VAR
	pRack 		: POINTER TO FB_Rack;
	pReactor 	: POINTER TO FB_Reactor;
	pNeedle		: POINTER TO FB_Needle; 
	pSlot 		: POINTER TO FB_PieceSlot;
	pTarget 	: POINTER TO FB_TargetBase;
	pPieceEx	: POINTER TO FB_PieceBase;
END_VAR
CASE refActionData.eAction OF
	E_Action.ACTION_ExchangePiece:
		pTarget := fbObjectDirectory.M_GetObjPointer(refActionData.nTarget);
		//Piece, welches gehandelt wird
		pPieceEx := pCorrelObject;
		//Welches Piece soll gehandelt werden?
		IF refActionData.aParams[2] = 0 THEN //Drop
			IF pPiece = 0 THEN
				M_CheckAction := E_ErrorIdCmd.ERRORID_NoPieceOnTool;
				RETURN;	
			END_IF
			//Luer kann folgende Pieces handeln
			//Tip, Needle, Septum in Verbindung mit Needle
			IF pPiece^.P_eObjectType = E_ObjectType.OBJECTTYPE_Tip THEN
				//Target muss TipRack sein
				IF pTarget^.P_eObjectType <> E_ObjectType.OBJECTTYPE_TipRack THEN
					M_CheckAction := E_ErrorIdCmd.ERRORID_UnsuitableTarget;
					RETURN;
				END_IF
			ELSIF pPiece^.P_eObjectType = E_ObjectType.OBJECTTYPE_Needle THEN
				pNeedle := pPiece;
				IF pNeedle^.P_pSeptum > 0 THEN
					//Target muss SeptumWaste sein
					IF pTarget^.P_eObjectType <> E_ObjectType.OBJECTTYPE_SeptumWaste THEN
						M_CheckAction := E_ErrorIdCmd.ERRORID_UnsuitableTarget;
						RETURN;
					END_IF
				ELSE
					//Target muss NeedleRack sein
					IF pTarget^.P_eObjectType <> E_ObjectType.OBJECTTYPE_NeedleRack THEN
						M_CheckAction := E_ErrorIdCmd.ERRORID_UnsuitableTarget;
						RETURN;
					END_IF
				END_IF
			ELSE
				M_CheckAction := E_ErrorIdCmd.ERRORID_InvalidPieceType;
				RETURN;
			END_IF
		ELSE //Take
			//Schon ein Piece am Tool?
			IF pPiece > 0 THEN
				IF pPiece^.P_eObjectType = E_ObjectType.OBJECTTYPE_Needle THEN
					pNeedle := pPiece;
					IF pNeedle^.P_pSeptum > 0 THEN
						M_CheckAction := E_ErrorIdCmd.ERRORID_PieceAlreadyOnTool;
						RETURN;
					ELSE
						//Target muss Reactor sein!
						IF pTarget^.P_eObjectType = E_ObjectType.OBJECTTYPE_Reactor THEN
							//Im Reaktor muss ein Vial und auf diesem sich ein Septum befinden
							pReactor := pTarget;
							IF pReactor^.P_pVial > 0 THEN
								IF pReactor^.P_pVial^.P_pSeptum = 0 THEN
									M_CheckAction := E_ErrorIdCmd.ERRORID_NoPieceInSlot;
									RETURN;
								END_IF
							ELSE
								M_CheckAction := E_ErrorIdCmd.ERRORID_NoPieceInSlot;
								RETURN;
							END_IF
						ELSE
							M_CheckAction := E_ErrorIdCmd.ERRORID_UnsuitableTarget;
							RETURN;
						END_IF
					END_IF
				ELSE
					M_CheckAction := E_ErrorIdCmd.ERRORID_PieceAlreadyOnTool;
					RETURN;
				END_IF
			ELSE 
				IF pPieceEx^.P_eObjectType = E_ObjectType.OBJECTTYPE_Septum THEN
					M_CheckAction := E_ErrorIdCmd.ERRORID_NoNeedleOnTool;
					RETURN;
				END_IF
			END_IF
		END_IF	
	E_Action.ACTION_DockTool:
		pTarget := fbObjectDirectory.M_GetObjPointer(refActionData.nTarget);
		//Piece am Tool?
		IF THIS^.pPiece > 0 THEN
			M_CheckAction := E_ErrorIdCmd.ERRORID_PieceAlreadyOnTool;
			RETURN;
		END_IF
		//Luer kann an PortRack andocken
		IF pTarget^.P_eObjectType = E_ObjectType.OBJECTTYPE_PortRack THEN
			pRack := pTarget;
			pSlot := pRack^.M_GetSlot(DINT_TO_UINT(refActionData.aParams[2]));
			IF pSlot > 0 THEN
				IF pSlot^.P_pPiece = 0 THEN
					M_CheckAction := E_ErrorIdCmd.ERRORID_NoPieceInSlot;
					RETURN;	
				END_IF
			ELSE
				M_CheckAction := E_ErrorIdCmd.ERRORID_InvalidTargetSlot;
				RETURN;
			END_IF
			//Im Slot muss ein Port sein
		ELSE
			M_CheckAction := E_ErrorIdCmd.ERRORID_UnsuitableTarget;
			RETURN;		
		END_IF
	E_Action.ACTION_MeasureTool:
		IF fbObjectDirectory.M_GetObjType(refActionData.nTarget) <> E_ObjectType.OBJECTTYPE_TipCalibrator THEN
			M_CheckAction := E_ErrorIdCmd.ERRORID_UnsuitableTarget;
			RETURN;
		END_IF
	E_Action.ACTION_InsertTool:
		IF pPiece = 0 THEN
			M_CheckAction := E_ErrorIdCmd.ERRORID_NoPieceOnTool;
		END_IF
	E_Action.ACTION_WashTool:
		//Washmode checken
		IF refActionData.aParams[2] = E_WashMode.MODE_WashInside THEN
			M_CheckAction := M_CheckBottles();
		ELSIF refActionData.aParams[2] = E_WashMode.MODE_WashOutside THEN
			;
		ELSIF refActionData.aParams[2] = E_WashMode.MODE_WashInOutside THEN
			M_CheckAction := M_CheckBottles();
		ELSE
			M_CheckAction := E_ErrorIdCmd.ERRORID_InvalidWashMode;	
		END_IF	
	E_Action.ACTION_Dispense, //BasicAction für ActionOnArray
	E_Action.ACTION_DryToolInside,
	E_Action.ACTION_TeachTarget:
		RETURN;
ELSE
	M_CheckAction := SUPER^.M_CheckAction(refActionData, pCorrelObject);
END_CASE
END_METHOD

METHOD M_CheckBottles : ERRORID
VAR_INPUT
END_VAR
IF pDiluter > 0 THEN
	M_CheckBottles := pDiluter^.M_CheckBottles(0);
END_IF
END_METHOD

METHOD M_CheckProps : ERRORID
VAR_INPUT
END_VAR
M_CheckProps := SUPER^.M_CheckProps();
IF M_CheckProps > 0 THEN
	RETURN;
END_IF
//Konfigurierte Properties checken
//zugeordneter Diluter
IF fbObjectDirectory.M_GetObjType(nDiluterObjId) <> E_ObjectType.OBJECTTYPE_Diluter THEN
	M_CheckProps := E_ErrorIdObjMgmt.ERRORID_InvalidDiluterObjId; //Error
	RETURN;
ELSE
	pDiluter := fbObjectDirectory.M_GetObjPointer(nDiluterObjId);
END_IF
END_METHOD

METHOD M_ClearAllProps
VAR_INPUT
	bIgnoreParent : BOOL; //Es wird das gesamte OD gelöscht. -> Zeiger auf Parent nicht mehr gültig!
END_VAR
pPneuChannelSyntGas := 0;
SUPER^.M_ClearAllProps(bIgnoreParent);
END_METHOD

METHOD M_ExeAction : ERRORID
VAR_INPUT
	refActionData : REFERENCE TO ST_ActionData;	
END_VAR
IF NOT (eCurrentState = E_MachineState.MACHINESTATE_Idle OR
	eCurrentState = E_MachineState.MACHINESTATE_Active OR
	eCurrentState = E_MachineState.MACHINESTATE_Ready) THEN
	M_ExeAction := E_ErrorIdCmd.ERRORID_InvalidState;
	RETURN;
END_IF

CASE refActionData.eAction OF
	
	E_Action.ACTION_Aspirate:
		IF NOT bAspirate THEN
			M_ExeAction := pDiluter^.M_CheckBottles(0); //Checken, ob Bottles OK
			IF M_ExeAction > 0 THEN
				RETURN;
			END_IF			
			nQuantity := refActionData.aParams[1];
			nFlow := refActionData.aParams[2];
			fbList.A_AddHeadValue( hList := hList, putValue := E_Action.ACTION_Aspirate);
			bAspirate := TRUE;
		END_IF
		
	E_Action.ACTION_Dispense:
		IF NOT bDispense THEN
			M_ExeAction := pDiluter^.M_CheckBottles(0); //Checken, ob Bottles OK
			IF M_ExeAction > 0 THEN
				RETURN;
			END_IF			
			nQuantity := refActionData.aParams[1];
			nFlow := refActionData.aParams[2];
			fbList.A_AddHeadValue(hList := hList, putValue := E_Action.ACTION_Dispense);
			bDispense := TRUE;
		END_IF
		
	E_Action.ACTION_Mix:
		IF NOT bMix THEN
			M_ExeAction := pDiluter^.M_CheckBottles(0); //Checken, ob Bottles OK
			IF M_ExeAction > 0 THEN
				RETURN;
			END_IF			
			nQuantity := refActionData.aParams[1];
			nFlowAsp := refActionData.aParams[2];
			nFlowDisp := refActionData.aParams[3];
			nMixRepeats := DINT_TO_UINT(refActionData.aParams[4]);
			nCurrMixRepeats := 0;
			tMixDelay1 := DINT_TO_TIME(refActionData.aParams[5]);
			tMixDelay2 := DINT_TO_TIME(refActionData.aParams[6]);
			fbList.A_AddHeadValue(hList := hList, putValue := E_Action.ACTION_Mix);
			bMix := TRUE;
		END_IF		
		
	E_Action.ACTION_Eject:
		//TipEjector vorhanden??
		IF pZAxisRef^.eFixedToolType <> E_MzToolType.TOOL_TYPE_TipEjector THEN
			M_ExeAction := 21212;
			RETURN;	
		END_IF
		
		IF NOT bEject THEN
			fbList.A_AddHeadValue(hList := hList, putValue := E_Action.ACTION_Eject);
			bEject := TRUE;
		END_IF
			
	E_Action.ACTION_SetPressure:
		fbSetPress(bExecute:= FALSE, pPneuChannelRef:= pPneuChannelSyntGas); //eventueller Fehler wird auch zurückgesetzt
		fbSetPress.bAwait := DINT_TO_BOOL(refActionData.aParams[1]);
		fbSetPress.nValue := DINT_TO_INT(refActionData.aParams[2]);
		fbSetPress.nTolerancePlus := DINT_TO_INT(refActionData.aParams[3]);
		fbSetPress.nToleranceMinus := DINT_TO_INT(refActionData.aParams[4]);
		fbSetPress.tTimeout := DINT_TO_TIME(refActionData.aParams[5]);
		
		fbSetPress(bExecute:= TRUE,	pPneuChannelRef:= pPneuChannelSyntGas, nErrorId=> M_ExeAction);
		IF fbSetPress.bError THEN
			RETURN;
		END_IF
		
		IF NOT bSetPress AND fbSetPress.bBusy THEN
			bSetPress := TRUE;
			fbList.A_AddHeadValue(hList := hList, putValue := E_Action.ACTION_SetPressure);
		ELSE
			RETURN;	
		END_IF
		
	E_Action.ACTION_SwitchPressure:
		eSwitchPressCtrl := DINT_TO_USINT(refActionData.aParams[1]);
		tPressTime := DINT_TO_TIME(refActionData.aParams[2]);
		//Wenn Aktion aktiv kann es sein das die Zeit noch läuft oder der Druck an ist
		IF bSwitchPress THEN	//Aktion ist aktiv
			IF eSwitchPressCtrl = E_PressCtrl.PRESSCTRL_PressOn THEN
				//Statemachine zurücksetzen
				nStateA_SwitchPress := 0;		
			ELSE
				aValves[nValveNrSynthGas].M_Off();
				nStateA_SwitchPress := 80;
			END_IF
		ELSE	//Aktion ist nicht aktiv
			IF eSwitchPressCtrl = E_PressCtrl.PRESSCTRL_PressOn THEN
				bSwitchPress := TRUE;
				fbList.A_AddHeadValue(hList := hList, putValue := E_Action.ACTION_SwitchPressure);
			ELSE
				aValves[nValveNrSynthGas].M_Off();
			END_IF
		END_IF
	ELSE
		M_ExeAction := SUPER^.M_ExeAction(refActionData);
		RETURN;
END_CASE

bBusy := TRUE;
eCurrentState := E_MachineState.MACHINESTATE_Active;
END_METHOD

METHOD M_GetAllProps : ERRORID
VAR_INPUT
	refCmdData : REFERENCE TO  ST_CmdData;
END_VAR
//BaseProperties lesen
SUPER^.M_GetAllProps(refCmdData);
//BaseProperties lesen
nCurrentPropIndex := nCurrentPropIndex + 1;
refCmdData.n32Data[nCurrentPropIndex] := nDiluterObjId;
nCurrentPropIndex := nCurrentPropIndex + 1;
refCmdData.n32Data[nCurrentPropIndex] := nDiluterObjId2;
nCurrentPropIndex := nCurrentPropIndex + 1;
refCmdData.n32Data[nCurrentPropIndex] := nDrypadArea;
nCurrentPropIndex := nCurrentPropIndex + 1;
refCmdData.n32Data[nCurrentPropIndex] := TIME_TO_DINT(tDryTime);
//TipEjector exist
nCurrentPropIndex := nCurrentPropIndex + 1;
IF pZAxisRef^.eFixedToolType = E_MzToolType.TOOL_TYPE_TipEjector THEN
	refCmdData.n32Data[nCurrentPropIndex] := 1;
ELSE
	refCmdData.n32Data[nCurrentPropIndex] := 0;
END_IF

nCurrentPropIndex := nCurrentPropIndex + 1;
IF pPneuChannelSyntGas > 0 THEN
	refCmdData.n32Data[nCurrentPropIndex] := pPneuChannelSyntGas^.nChannel;	
ELSE
	refCmdData.n32Data[nCurrentPropIndex] := 0;
END_IF

nCurrentPropIndex := nCurrentPropIndex + 1;
refCmdData.n32Data[nCurrentPropIndex] := nValveNrSynthGas;
nCurrentPropIndex := nCurrentPropIndex + 1;
refCmdData.n32Data[nCurrentPropIndex] := nValveNrDiluter;
nCurrentPropIndex := nCurrentPropIndex + 1;
refCmdData.n32Data[nCurrentPropIndex] := nValveNrLuer;
nCurrentPropIndex := nCurrentPropIndex + 1;
refCmdData.n32Data[nCurrentPropIndex] := REAL_TO_DINT(rDockOffset);
nCurrentPropIndex := nCurrentPropIndex + 1;
refCmdData.n32Data[nCurrentPropIndex] := nDispFlowFix;
END_METHOD

METHOD M_SetAllProps : ERRORID
VAR_INPUT
	refCmdData : REFERENCE TO  ST_CmdData;
END_VAR

VAR
	nPneuChannel : USINT;
END_VAR
M_SetAllProps := SUPER^.M_SetAllProps(refCmdData);

IF M_SetAllProps > 0 THEN
	RETURN;
END_IF

//Diluter 1 (SingleDiluter)
nCurrentPropIndex := nCurrentPropIndex + 1;
nSpecPropIndex := nCurrentPropIndex;
nDiluterObjId :=  DINT_TO_UINT(refCmdData.n32Data[nCurrentPropIndex]);

IF fbObjectDirectory.M_GetObjType(nDiluterObjId) = E_ObjectType.OBJECTTYPE_Diluter THEN
	pDiluter := fbObjectDirectory.M_GetObjPointer(nDiluterObjId);
ELSE
	M_SetAllProps := E_ErrorIdObjMgmt.ERRORID_InvalidDiluterObjId;
	RETURN;
END_IF

//Diluter 2 (TwinDiluter)
nCurrentPropIndex := nCurrentPropIndex + 1;
nDiluterObjId2 :=  DINT_TO_UINT(refCmdData.n32Data[nCurrentPropIndex]);

nCurrentPropIndex := nCurrentPropIndex + 1;
nDrypadArea := DINT_TO_USINT(refCmdData.n32Data[nCurrentPropIndex]);
nCurrentPropIndex := nCurrentPropIndex + 1;
tDryTime := DINT_TO_TIME(refCmdData.n32Data[nCurrentPropIndex]);

//TipEjector
nCurrentPropIndex := nCurrentPropIndex + 1;
IF refCmdData.n32Data[nCurrentPropIndex].0 THEN
	pZAxisRef^.eFixedToolType := E_MzToolType.TOOL_TYPE_TipEjector;
ELSE
	pZAxisRef^.eFixedToolType := E_MzToolType.TOOL_TYPE_None;
END_IF

nCurrentPropIndex := nCurrentPropIndex + 1;
nPneuChannel := DINT_TO_USINT(refCmdData.n32Data[nCurrentPropIndex]);
IF NOT (nPneuChannel > 0 AND nPneuChannel <= cNoOfPneuChannels) THEN
	M_SetAllProps := E_ErrorIdObjMgmt.ERRORID_InvalidPneuChannel;
	RETURN;
END_IF
pPneuChannelSyntGas := ADR(aFbPneuChannel[nPneuChannel]);

nCurrentPropIndex := nCurrentPropIndex + 1;
nValveNrSynthGas := DINT_TO_USINT(refCmdData.n32Data[nCurrentPropIndex]);
IF NOT(nValveNrSynthGas >= 0 AND nValveNrSynthGas <= cNoOfValves) THEN
	M_SetAllProps := E_ErrorIdObjMgmt.ERRORID_InvalidValveNumber;
	RETURN;
END_IF

nCurrentPropIndex := nCurrentPropIndex + 1;
nValveNrDiluter := DINT_TO_USINT(refCmdData.n32Data[nCurrentPropIndex]);
IF NOT(nValveNrDiluter >= 0 AND nValveNrDiluter <= cNoOfValves) THEN
	M_SetAllProps := E_ErrorIdObjMgmt.ERRORID_InvalidValveNumber;
END_IF

nCurrentPropIndex := nCurrentPropIndex + 1;
nValveNrLuer := DINT_TO_USINT(refCmdData.n32Data[nCurrentPropIndex]);
IF NOT(nValveNrLuer >= 0 AND nValveNrLuer <= cNoOfValves) THEN
	M_SetAllProps := E_ErrorIdObjMgmt.ERRORID_InvalidValveNumber;
END_IF

nCurrentPropIndex := nCurrentPropIndex + 1;
rDockOffset := DINT_TO_REAL(refCmdData.n32Data[nCurrentPropIndex]);

//DispFlowFix
nCurrentPropIndex := nCurrentPropIndex + 1;
nDispFlowFix := refCmdData.n32Data[nCurrentPropIndex];

nNoOfProps := nCurrentPropIndex + 1;
END_METHOD

METHOD M_SetPrintParams : ST_MethResult
VAR_INPUT
	eType 		: E_PrintParamType;
	nNumerator	: USINT;
	nValue		: DINT;
END_VAR
IF eType = E_PrintParamType.Flow THEN
	IF nNumerator <> 1 THEN
		M_SetPrintParams.bError := TRUE;
		M_SetPrintParams.nErrorId := E_ErrorIdCmd.ERRORID_InvalidPrintParamNumerator;
		RETURN;
	END_IF
	fbObjectDirectory.M_SetObjChange(nObjectID); //Info an GUI
	nDispFlowFix := nValue;
ELSE
	M_SetPrintParams.bError := TRUE;
	M_SetPrintParams.nErrorId := E_ErrorIdCmd.ERRORID_InvalidPrintParamType;
END_IF
END_METHOD

METHOD M_SetSingleProp : ERRORID
VAR_INPUT
	refCmdData : REFERENCE TO  ST_CmdData;
END_VAR

VAR
	nPneuChannel : USINT;
END_VAR
IF nSpecPropIndex + 5 = refCmdData.aHeader[1] THEN	//PneuChannelSynthGas
	nPneuChannel := DINT_TO_USINT(refCmdData.n32Data[0]);
	IF NOT (nPneuChannel > 0 AND nPneuChannel <= cNoOfPneuChannels) THEN
		M_SetSingleProp := E_ErrorIdObjMgmt.ERRORID_InvalidPneuChannel;
		RETURN;	
	END_IF
	pPneuChannelSyntGas := ADR(aFbPneuChannel[nPneuChannel]);
ELSIF nSpecPropIndex + 6 = refCmdData.aHeader[1] THEN	//ValveSynthGas
	IF refCmdData.n32Data[0] >= 0 AND refCmdData.n32Data[0] <= cNoOfValves THEN
		nValveNrSynthGas := DINT_TO_USINT(refCmdData.n32Data[0]);
	ELSE
		M_SetSingleProp := E_ErrorIdObjMgmt.ERRORID_InvalidValveNumber;
	END_IF
ELSIF nSpecPropIndex + 7 = refCmdData.aHeader[1] THEN	//ValveNrDiluter
	IF refCmdData.n32Data[0] >= 0 AND refCmdData.n32Data[0] <= cNoOfValves THEN
		nValveNrDiluter := DINT_TO_USINT(refCmdData.n32Data[0]);
	ELSE
		M_SetSingleProp := E_ErrorIdObjMgmt.ERRORID_InvalidValveNumber;
	END_IF	
ELSIF nSpecPropIndex + 8 = refCmdData.aHeader[1] THEN	//ValveNrLuer
	IF refCmdData.n32Data[0] >= 0 AND refCmdData.n32Data[0] <= cNoOfValves THEN
		nValveNrLuer := DINT_TO_USINT(refCmdData.n32Data[0]);
	ELSE
		M_SetSingleProp := E_ErrorIdObjMgmt.ERRORID_InvalidValveNumber;
	END_IF	
ELSIF nSpecPropIndex + 9 = refCmdData.aHeader[1] THEN	//DockOffset
	rDockOffset := DINT_TO_REAL(refCmdData.n32Data[0]);
ELSIF nSpecPropIndex + 10 = refCmdData.aHeader[1] THEN	//DispFlowFix
	nDispFlowFix := refCmdData.n32Data[0];
ELSE
	M_SetSingleProp := SUPER^.M_SetSingleProp(refCmdData);
END_IF
END_METHOD

METHOD M_StartUniDispense : ERRORID
VAR_INPUT
	nParam1 : DINT; //Quantity
	nParam2 : DINT; //unused
END_VAR

VAR_OUTPUT
	bIsContinous : BOOL;
END_VAR

VAR
	stActionData : ST_ActionData;
END_VAR
IF nParam1 = 0 THEN
	bIsContinous := TRUE;
	bEndless := TRUE;
ELSE
	bEndless := FALSE;
END_IF

stActionData.aParams[1] := nParam1; //Quantitiy
stActionData.aParams[2] := nDispFlowFix;
stActionData.eAction := E_Action.ACTION_Dispense;
M_StartUniDispense := M_ExeAction(stActionData);
END_METHOD

METHOD M_StopUniDispense : ERRORID
VAR_INPUT
END_VAR
M_CancelAction(E_Action.ACTION_Dispense);
END_METHOD

METHOD M_SwitchValveDiluter
VAR_INPUT
	bOn : BOOL;
END_VAR
IF nValveNrDiluter > 0 THEN
	IF bOn THEN
		aValves[nValveNrDiluter].M_On(1);
	ELSE
		aValves[nValveNrDiluter].M_Off();
	END_IF
END_IF
END_METHOD

METHOD M_SwitchValveLuer
VAR_INPUT
	bOn : BOOL;
END_VAR
IF nValveNrLuer > 0 THEN
	IF bOn THEN
		aValves[nValveNrLuer].M_On(1);
	ELSE
		aValves[nValveNrLuer].M_Off();
	END_IF
END_IF
END_METHOD

METHOD M_SwitchValveSynthGas
VAR_INPUT
	bOn : BOOL;
END_VAR
IF nValveNrSynthGas > 0 THEN
	IF bOn THEN
		aValves[nValveNrSynthGas].M_On(1);
	ELSE
		aValves[nValveNrSynthGas].M_Off();
	END_IF
END_IF
END_METHOD

PROPERTY P_nDrypadArea : USINT
GET
P_nDrypadArea := nDrypadArea;
END_GET
END_PROPERTY

PROPERTY P_pDiluter : POINTER TO FB_DILUTER
GET
P_pDiluter := pDiluter;
END_GET
END_PROPERTY

PROPERTY P_rDockOffset : REAL
GET
P_rDockOffset := rDockOffset;
END_GET
END_PROPERTY

PROPERTY P_stAbsPosPhys : ST_3DPoint
GET
VAR
	stTemp	: ST_3DPoint;
	stDim	: ST_3DDimension;
END_VAR
//Die absolute Postion eines Tool in "Z" hat nicht den gleichen Bezug wie X und Y
//X und Y beziehen sich auf den Koordinatenursprung, wenn die Achsen theoretischn aus Antrieb (0;0) stehen
//Z bezieht sich auf die Sliderunterkante des Z-Antriebes verechnet mit AbsPos vom Head(Ergebnis ist in den meisten Fällen negativ)

//Offset und RelPos addieren
stTemp := F_Add3DPoints(stRelPos,stOffset);

//Offsets der Pieces verrechnen
IF pPiece > 0 THEN
	stDim := pPiece^.P_stDimension;
	IF NOT pPiece^.P_bIgnoreOffset THEN
		stTemp := F_Add3DPoints(stTemp,pPiece^.P_stOffset);	
	END_IF
	stTemp.Z := stTemp.Z + pPiece^.P_rZOverlapTool - stDim.Height;
END_IF

//AbsPos vom ParentSlot holen
IF pParentSlot > 0 THEN
	stTemp := F_Add3DPoints(stTemp,pParentSlot^.P_stAbsPos);	
END_IF
P_stAbsPosPhys := stTemp;
END_GET
END_PROPERTY

PROPERTY P_stCurrentXYArea : FB_RectAngle
GET
VAR
	stPoint : ST_3DPoint;
	stDim	: ST_3DDimension;
END_VAR
stPoint := P_stCurrentPosPhys;
IF pPiece > 0 THEN
	stDim := pPiece^.P_stDimension;
	P_stCurrentXYArea.X1 := stPoint.X - stDim.Width / 2.0;
	P_stCurrentXYArea.X2 := stPoint.X + stDim.Width / 2.0;
	P_stCurrentXYArea.Y1 := stPoint.Y - stDim.Width / 2.0;
	P_stCurrentXYArea.Y2 := stPoint.Y + stDim.Width / 2.0;
ELSE
	P_stCurrentXYArea.X1 := stPoint.X - 2000.0;
	P_stCurrentXYArea.X2 := stPoint.X + 2000.0;
	P_stCurrentXYArea.Y1 := stPoint.Y - 2000.0;
	P_stCurrentXYArea.Y2 := stPoint.Y + 2000.0;	
END_IF
END_GET
END_PROPERTY

PROPERTY P_tDryTime : TIME
GET
P_tDryTime := tDryTime;
END_GET
END_PROPERTY

END_FUNCTION_BLOCK

// ---- Objects/Tools/FB_VacuumHandler.TcPOU
FUNCTION_BLOCK FB_VacuumHandler EXTENDS FB_MzTool
VAR_INPUT
END_VAR
VAR_OUTPUT
END_VAR
VAR
	

	//SpecProperties
	pPneuChannelVac		: POINTER TO FB_PneuChannelRef;
	nValveNrVacuum		: USINT;
	nHoldVacuumVial		: INT;
	nHoldVacuumSeptum	: INT;
	rDockOffset			: REAL;

	//****************************************Aktionvariablen****************************************************
	
	stActionDataSpec	: ST_ActionData;
	
	//Action: "InitSpec"
	bInitSpec			: BOOL;
	bInitSpecFlag		: BOOL := TRUE;
	nStateA_InitSpec	: USINT;
	
	//Action: "SetVacuum"
	bSetVacuum			: BOOL;
	fbSetVacuum			: FB_SetPressure;
	
	//Action: "SwitchPressure"
	bSwitchPress		: BOOL;			
	nStateA_SwitchPress	: USINT;		//State von A_SwitchPress()
	nSwitchPressChannel	: USINT;
	eSwitchPressCtrl	: E_PressCtrl;
	tPressTime			: TIME;			//nach dieser Zeit Ventil automatisch wieder zu
	timerPress			: TON;			//Timer für Öffnungszeit Druckventil 		
	
END_VAR

IF eCurrentState = E_MachineState.MACHINESTATE_Active THEN
	
	IF bSetVacuum THEN
		fbSetVacuum(pPneuChannelRef:= pPneuChannelVac);
		IF NOT fbSetVacuum.bBusy THEN
			IF fbSetVacuum.bError THEN
				bError := TRUE;
				stError.ErrorId := fbSetVacuum.nErrorId;
				stError.POU := E_POU.POU_FB_VacuumHandler;
				fbErrorList.M_Add(stError);
			END_IF
			bSetVacuum := FALSE;
			fbSetVacuum(pPneuChannelRef:= pPneuChannelVac, bExecute:= FALSE);
			M_RemoveListEntry(nSearchValue:= E_Action.ACTION_SetVacuum);
		END_IF
	END_IF	
	
	IF bSwitchPress THEN	//Kartuschendruck einstellen und Ein-bzw. Aus schalten 
		A_SwitchPress();
		IF nStateA_SwitchPress >= 80 THEN
			IF nStateA_SwitchPress >= 99 THEN
				bError := TRUE;
			END_IF
			bSwitchPress := FALSE;
			nStateA_SwitchPress := 0;
			M_RemoveListEntry(nSearchValue:= E_Action.ACTION_SwitchPressure);
		END_IF
	END_IF	
END_IF

SUPER^();	//FB_MzTool aufrufen

//Prozessdaten aktualisieren
IF pPneuChannelVac > 0 THEN
	stProcessData.n32Data[7] := pPneuChannelVac^.P_nCurrentPressure;
END_IF

IF nValveNrVacuum > 0 THEN
	IF aValves[nValveNrVacuum].bDigiOut1 THEN
		stProcessData.n32Data[8] := E_PressCtrl.PRESSCTRL_VacOn;
	ELSE
		stProcessData.n32Data[8] := E_PressCtrl.PRESSCTRL_Off;
	END_IF
END_IF

aObjProcData[nNotifyId] := stProcessData;

ACTION A_Reset:
//Ist noch eine Aktion aktiv?
IF nStateA_ResetSpec = 0 THEN 
	nStateA_ResetSpec := 80;
END_IF

SUPER^.A_Reset();
END_ACTION

ACTION A_Stop:
IF nStateA_Stop = 0 THEN
	nStateA_Stop := 1;
END_IF

SUPER^.A_Stop();
END_ACTION

ACTION A_SwitchPress:
CASE nStateA_SwitchPress OF
	0:	//Ventil Einschalten
		IF eSwitchPressCtrl = E_PressCtrl.PRESSCTRL_PressOn OR eSwitchPressCtrl = E_PressCtrl.PRESSCTRL_VacOn THEN
			aValves[M_GetValveNr(nSwitchPressChannel)].M_On(1);
		END_IF
	
		//Timer starten
		IF tPressTime = T#0S THEN
			nStateA_SwitchPress := 80;
			RETURN;	
		END_IF
		
		timerPress(IN:= FALSE);
		timerPress(IN:= TRUE, PT:= tPressTime);
		nStateA_SwitchPress := 1;
		
	1:	//Warten bis Zeitabgelaufen
		timerPress();
		IF timerPress.Q THEN
			timerPress(IN:= FALSE);
			aValves[M_GetValveNr(nSwitchPressChannel)].M_Off();
			nStateA_SwitchPress := 80;
		END_IF
		
	70:	//Abbrechen
		timerPress(IN:= FALSE);
		aValves[M_GetValveNr(nSwitchPressChannel)].M_Off();
		nStateA_SwitchPress := 80;
END_CASE
END_ACTION

METHOD FB_init : BOOL
VAR_INPUT
	bInitRetains : BOOL; // if TRUE, the retain variables are initialized (warm start / cold start)
	bInCopyCode : BOOL;  // if TRUE, the instance afterwards gets moved into the copy code (online change)
END_VAR
eObjectType := E_ObjectType.OBJECTTYPE_VacuumHandler;
eObjectGroup := E_ObjectGroup.OBJECTGROUP_MzTool OR E_ObjectGroup.OBJECTGROUP_Device;
END_METHOD

METHOD M_AddChild : ERRORID
VAR_INPUT
	pObject : POINTER TO FB_Object;
	nSlotNr	: UINT;
	nIndex 	: INT;	
END_VAR
//Kann folgende Objekt-Typen aufnehmen
//Vial, Septum
IF pObject > 0 THEN
	IF pObject^.P_eObjectType = E_ObjectType.OBJECTTYPE_Vial OR
		pObject^.P_eObjectType = E_ObjectType.OBJECTTYPE_Septum THEN
		M_AddChild := SUPER^.M_AddChild(pObject,nSlotNr,nIndex);
	ELSE
		M_AddChild := E_ErrorIdObjMgmt.ERRORID_InvalidParentObject;
	END_IF
ELSE
	M_AddChild := E_ErrorIdObjMgmt.ERRORID_InvalidParentObject;
END_IF
END_METHOD

METHOD M_CancelAction
VAR_INPUT
	eAction : E_Action;
END_VAR
CASE eAction OF

	E_Action.ACTION_SetVacuum:
		IF bSetVacuum THEN
			fbSetVacuum(bExecute:= FALSE, pPneuChannelRef:= pPneuChannelVac);
		END_IF

	E_Action.ACTION_SwitchPressure:
		IF bSwitchPress AND nStateA_SwitchPress < 70 THEN
			nStateA_SwitchPress := 70;
		END_IF	
ELSE
	SUPER^.M_CancelAction(eAction);
END_CASE
END_METHOD

METHOD M_CheckAction : ERRORID
VAR_INPUT
	refActionData 	: REFERENCE TO ST_ActionData;
	pCorrelObject	: POINTER TO FB_Object;
END_VAR

VAR
	pRack : POINTER TO FB_Rack;
	pReactor : POINTER TO FB_Reactor;
	pSlot : POINTER TO FB_PieceSlot;
	pTarget : POINTER TO FB_TargetBase;
END_VAR
CASE refActionData.eAction OF
	E_Action.ACTION_ExchangePiece:
		pTarget := fbObjectDirectory.M_GetObjPointer(refActionData.nTarget);
		//Welches Piece soll gehandelt werden?
		IF refActionData.aParams[2] = 0 THEN //Drop
			IF pPiece = 0 THEN
				M_CheckAction := E_ErrorIdCmd.ERRORID_NoPieceOnTool;
				RETURN;	
			END_IF
			//VacuumHandler kann folgende Pieces handeln
			//Vial, Septum
			IF pPiece^.P_eObjectType = E_ObjectType.OBJECTTYPE_Vial THEN
				//Target muss VialRack oder Reaktor sein
				IF pTarget^.P_eObjectType = E_ObjectType.OBJECTTYPE_VialRack THEN
					pRack := pTarget;
					//Slot muss frei sein
					pSlot := pRack^.M_GetSlot(DINT_TO_UINT(refActionData.aParams[1]));
					IF pSlot = 0 THEN
						M_CheckAction := E_ErrorIdCmd.ERRORID_InvalidTargetSlot;
						RETURN;
					ELSIF pSlot^.P_pPiece > 0 THEN
						M_CheckAction := E_ErrorIdCmd.ERRORID_PieceAlreadyInSlot;
						RETURN;
					END_IF
				ELSIF pTarget^.P_eObjectType = E_ObjectType.OBJECTTYPE_Reactor THEN
					//Slot muss frei sein
					//Hier kann ein Vial geholt werden
					pReactor := pTarget;
					IF pReactor^.P_pVial > 0 THEN
						M_CheckAction := E_ErrorIdCmd.ERRORID_PieceAlreadyInSlot;
						RETURN;
					END_IF
				ELSE
					M_CheckAction := E_ErrorIdCmd.ERRORID_UnsuitableTarget;
					RETURN;
				END_IF
			ELSIF pPiece^.P_eObjectType = E_ObjectType.OBJECTTYPE_Septum THEN
				//Target kann nur Reaktor mit Vial sein
				//Ob ein Vial im Reaktor steht, wird in FB_Reactor.M_CheckActon() geprüft 
				IF pTarget^.P_eObjectType <> E_ObjectType.OBJECTTYPE_Reactor THEN 
					M_CheckAction := E_ErrorIdCmd.ERRORID_UnsuitableTarget;
					RETURN;
				END_IF
			ELSE
				M_CheckAction := E_ErrorIdCmd.ERRORID_InvalidPieceType;
				RETURN;
			END_IF
		ELSE  //Take
			//Schon ein Piece am Tool?
			IF THIS^.pPiece > 0 THEN
				M_CheckAction := E_ErrorIdCmd.ERRORID_PieceAlreadyOnTool;
				RETURN;
			END_IF
			
			IF pTarget^.P_eObjectType = E_ObjectType.OBJECTTYPE_Reactor THEN
				//Hier kann ein Vial geholt werden
				pReactor := pTarget;
				IF pReactor^.P_pVial = 0 THEN
					M_CheckAction := E_ErrorIdCmd.ERRORID_NoPieceInSlot;
					RETURN;
				ELSIF pReactor^.P_pVial^.P_pSeptum > 0 THEN
					M_CheckAction := E_ErrorIdCmd.ERRORID_SeptumAlreadyOnVial;
					RETURN;
				END_IF
			ELSIF pTarget^.P_eObjectType = E_ObjectType.OBJECTTYPE_VialRack THEN
				//Hier kann ein Vial geholt werden
				pRack := pTarget;
				pSlot := pRack^.M_GetSlot(DINT_TO_UINT(refActionData.aParams[1]));
				IF pSlot > 0 THEN
					IF pSlot^.P_pPiece = 0 THEN
						M_CheckAction := E_ErrorIdCmd.ERRORID_NoPieceInSlot;
						RETURN;
					ELSIF pSlot^.P_pPiece^.P_eObjectType <> E_ObjectType.OBJECTTYPE_Vial THEN
						M_CheckAction := E_ErrorIdCmd.ERRORID_InvalidPieceType;
						RETURN;
					END_IF
				ELSE
					M_CheckAction := E_ErrorIdCmd.ERRORID_InvalidTargetSlot;
					RETURN;				
				END_IF		
			ELSIF pTarget^.P_eObjectType = E_ObjectType.OBJECTTYPE_SeptumRack THEN
				//Hier kann ein Septum geholt werden 
				pRack := pTarget;
				pSlot := pRack^.M_GetSlot(DINT_TO_UINT(refActionData.aParams[1]));
				IF pSlot > 0 THEN
					IF pSlot^.P_pPiece = 0 THEN
						M_CheckAction := E_ErrorIdCmd.ERRORID_NoPieceInSlot;
						RETURN;
					ELSIF pSlot^.P_pPiece^.P_eObjectType <> E_ObjectType.OBJECTTYPE_Septum THEN
						M_CheckAction := E_ErrorIdCmd.ERRORID_InvalidPieceType;
						RETURN;
					END_IF
				ELSE
					M_CheckAction := E_ErrorIdCmd.ERRORID_InvalidTargetSlot;
					RETURN;				
				END_IF
			END_IF
		END_IF	
ELSE
	M_CheckAction := SUPER^.M_CheckAction(refActionData, pCorrelObject);
END_CASE
END_METHOD

METHOD M_ClearAllProps
VAR_INPUT
	bIgnoreParent : BOOL; //Es wird das gesamte OD gelöscht. -> Zeiger auf Parent nicht mehr gültig!
END_VAR
pPneuChannelVac := 0;
SUPER^.M_ClearAllProps(bIgnoreParent);
END_METHOD

METHOD M_ExeAction : ERRORID
VAR_INPUT
	refActionData : REFERENCE TO ST_ActionData;	
END_VAR
IF NOT (eCurrentState = E_MachineState.MACHINESTATE_Idle OR
	eCurrentState = E_MachineState.MACHINESTATE_Active OR
	eCurrentState = E_MachineState.MACHINESTATE_Ready) THEN
	M_ExeAction := E_ErrorIdCmd.ERRORID_InvalidState;
	RETURN;
END_IF

CASE refActionData.eAction OF
	E_Action.ACTION_SetVacuum:
		fbSetVacuum(bExecute:= FALSE, pPneuChannelRef:= pPneuChannelVac); //eventueller Fehler wird auch zurückgesetzt
		fbSetVacuum.bAwait := DINT_TO_BOOL(refActionData.aParams[1]);
		fbSetVacuum.nValue := DINT_TO_INT(refActionData.aParams[2]);
		fbSetVacuum.nTolerancePlus := DINT_TO_INT(refActionData.aParams[3]);
		fbSetVacuum.nToleranceMinus := DINT_TO_INT(refActionData.aParams[4]);
		fbSetVacuum.tTimeout := DINT_TO_TIME(refActionData.aParams[5]);
		
		fbSetVacuum(bExecute:= TRUE, pPneuChannelRef:= pPneuChannelVac,nErrorId=> M_ExeAction);
		IF fbSetVacuum.bError THEN
			RETURN;
		END_IF
		
		IF NOT bSetVacuum AND fbSetVacuum.bBusy THEN
			bSetVacuum := TRUE;
			fbList.A_AddHeadValue(hList := hList, putValue := E_Action.ACTION_SetVacuum);
		ELSE
			RETURN;	
		END_IF
		
	E_Action.ACTION_SwitchPressure:
		//Channel checken
		nSwitchPressChannel := DINT_TO_USINT(refActionData.aParams[1]);
		IF M_GetValveNr(nSwitchPressChannel) = 0 THEN
			M_ExeAction := E_ErrorIdObjMgmt.ERRORID_InvalidPneuChannel;
			RETURN;
		END_IF
		eSwitchPressCtrl := DINT_TO_USINT(refActionData.aParams[2]);
		tPressTime := DINT_TO_TIME(refActionData.aParams[3]);
		IF bSwitchPress THEN	//Aktion ist aktiv
			//Statemachine zurücksetzen
		 	nStateA_SwitchPress := 0;		
			aValves[M_GetValveNr(nSwitchPressChannel)].M_Off();
			nStateA_SwitchPress := 80;
		ELSE //Aktion ist nicht aktiv
			IF eSwitchPressCtrl = E_PressCtrl.PRESSCTRL_PressOn OR eSwitchPressCtrl = E_PressCtrl.PRESSCTRL_VacOn THEN
				bSwitchPress := TRUE;
				fbList.A_AddHeadValue(hList := hList, putValue := E_Action.ACTION_SwitchPressure);
			ELSE
				aValves[M_GetValveNr(nSwitchPressChannel)].M_Off();
			END_IF			
		END_IF
	ELSE
		M_ExeAction := SUPER^.M_ExeAction(refActionData);
		RETURN;
END_CASE

bBusy := TRUE;
eCurrentState := E_MachineState.MACHINESTATE_Active;
END_METHOD

METHOD M_GetAllProps : ERRORID
VAR_INPUT
	refCmdData : REFERENCE TO  ST_CmdData;
END_VAR
//BaseProperties lesen
SUPER^.M_GetAllProps(refCmdData);
nCurrentPropIndex := nCurrentPropIndex + 1;
IF pPneuChannelVac > 0 THEN
	refCmdData.n32Data[nCurrentPropIndex] := pPneuChannelVac^.nChannel;
ELSE
	refCmdData.n32Data[nCurrentPropIndex] := 0;
END_IF
nCurrentPropIndex := nCurrentPropIndex + 1;
refCmdData.n32Data[nCurrentPropIndex] := nValveNrVacuum;
nCurrentPropIndex := nCurrentPropIndex + 1;
refCmdData.n32Data[nCurrentPropIndex] := nHoldVacuumVial;
nCurrentPropIndex := nCurrentPropIndex + 1;
refCmdData.n32Data[nCurrentPropIndex] := nHoldVacuumSeptum;
nCurrentPropIndex := nCurrentPropIndex + 1;
refCmdData.n32Data[nCurrentPropIndex] := REAL_TO_DINT(rDockOffset);
END_METHOD

METHOD PRIVATE M_GetValveNr : USINT
VAR_INPUT
	nChannel : USINT;
END_VAR
IF nChannel = 1 THEN
	M_GetValveNr := nValveNrVacuum;
END_IF
END_METHOD

METHOD M_SetAllProps : ERRORID
VAR_INPUT
	refCmdData : REFERENCE TO  ST_CmdData;
END_VAR

VAR
	nPneuChannel : USINT;
END_VAR
M_SetAllProps := SUPER^.M_SetAllProps(refCmdData);

IF M_SetAllProps > 0 THEN
	RETURN;
END_IF

nCurrentPropIndex := nCurrentPropIndex + 1;
nSpecPropIndex := nCurrentPropIndex;
nPneuChannel := DINT_TO_USINT(refCmdData.n32Data[nCurrentPropIndex]);
IF NOT (nPneuChannel >= 0 AND nPneuChannel <= cNoOfPneuChannels) THEN
	M_SetAllProps := E_ErrorIdObjMgmt.ERRORID_InvalidPneuChannel;
	RETURN;	
END_IF
pPneuChannelVac := ADR(aFbPneuChannel[nPneuChannel]);

nCurrentPropIndex := nCurrentPropIndex + 1;
nValveNrVacuum := DINT_TO_USINT(refCmdData.n32Data[nCurrentPropIndex]);
IF NOT (nValveNrVacuum > 0 AND nValveNrVacuum <= cNoOfValves) THEN
	M_SetAllProps := E_ErrorIdObjMgmt.ERRORID_InvalidValveNumber;
	RETURN;
END_IF

nCurrentPropIndex := nCurrentPropIndex + 1;
nHoldVacuumVial := DINT_TO_INT(refCmdData.n32Data[nCurrentPropIndex]);

nCurrentPropIndex := nCurrentPropIndex + 1;
nHoldVacuumSeptum := DINT_TO_INT(refCmdData.n32Data[nCurrentPropIndex]);

nCurrentPropIndex := nCurrentPropIndex + 1;
rDockOffset := DINT_TO_REAL(refCmdData.n32Data[nCurrentPropIndex]);

nNoOfProps := nCurrentPropIndex + 1;
END_METHOD

METHOD M_SetSingleProp : ERRORID
VAR_INPUT
	refCmdData : REFERENCE TO  ST_CmdData;
END_VAR

VAR
	nPneuChannel : USINT;
END_VAR
IF nSpecPropIndex = refCmdData.aHeader[1] THEN	//PneuChannelVacuum
	nPneuChannel := DINT_TO_USINT(refCmdData.n32Data[0]);
	IF NOT (nPneuChannel > 0 AND nPneuChannel <= cNoOfPneuChannels) THEN
		M_SetSingleProp := E_ErrorIdObjMgmt.ERRORID_InvalidPneuChannel;
		RETURN;	
	END_IF
	pPneuChannelVac := ADR(aFbPneuChannel[nPneuChannel]);
ELSIF nSpecPropIndex + 1 = refCmdData.aHeader[1] THEN	//ValveNrVacuum
	IF refCmdData.n32Data[0] >= 0 AND refCmdData.n32Data[0] <= cNoOfValves THEN
		nValveNrVacuum := DINT_TO_USINT(refCmdData.n32Data[0]);
	ELSE
		M_SetSingleProp := E_ErrorIdObjMgmt.ERRORID_InvalidValveNumber;
	END_IF
ELSIF nSpecPropIndex + 2 = refCmdData.aHeader[1] THEN	//HoldVacVial
	nHoldVacuumVial := DINT_TO_INT(refCmdData.n32Data[0]);
ELSIF nSpecPropIndex + 3 = refCmdData.aHeader[1] THEN	//HoldVacSeptum
	nHoldVacuumSeptum := DINT_TO_INT(refCmdData.n32Data[0]);
ELSIF nSpecPropIndex + 4 = refCmdData.aHeader[1] THEN	//DockOffset
	rDockOffset := DINT_TO_REAL(refCmdData.n32Data[0]);
ELSE
	M_SetSingleProp := SUPER^.M_SetSingleProp(refCmdData);
END_IF
END_METHOD

PROPERTY P_nHoldVacSept : INT
GET
P_nHoldVacSept := nHoldVacuumSeptum;
END_GET
END_PROPERTY

PROPERTY P_nHoldVacVial : INT
GET
P_nHoldVacVial := nHoldVacuumVial;
END_GET
END_PROPERTY

PROPERTY P_rDockOffset : REAL
GET
P_rDockOffset := rDockOffset;
END_GET
END_PROPERTY

END_FUNCTION_BLOCK

// ---- Objects/Tools/FB_SolenoidPip.TcPOU
FUNCTION_BLOCK FB_SolenoidPip EXTENDS FB_GCodeTool IMPLEMENTS I_UsingDryPad
VAR_INPUT
END_VAR
VAR_OUTPUT
END_VAR
VAR
	//Specproperties
	nDiluterObjId		: UINT;
	pDiluter			: POINTER TO FB_Diluter;
	pPneuChannelPress	: POINTER TO FB_PneuChannelRef;
	
	nFrequency			: UINT;
	nPulse				: UINT;
	//PrePeakTime wird direkt in pPiezoRef gespeichert
	
	rAspFrequSweepStart		: REAL;
	rAspFrequSweepEnd 		: REAL;
	rAspFrequSweepTime		: REAL;
	nAspiratePulse			: UINT;
	
	rDispFrequSweepStart	: REAL;
	rDispFrequSweepEnd 		: REAL;
	rDispFrequSweepTime		: REAL;
	nDispensePulse			: UINT;
		
	nDrypadArea				: USINT;
	tDryTime				: TIME;
	pFbPiezoRef				: POINTER TO FB_PiezoRef;
	fbPiezoControl			: FB_PiezoControl;
	
	//****************************************Aktionvariablen****************************************************
	
	stActionDataSpec	: ST_ActionData;
	
	//Sweep
	rFrequStep			: REAL;
	//rFrequStart			: REAL;
	rFrequNew			: REAL;
	rSweepSteps			: REAL;
	rCurrentSweepStep	: REAL;
	
	
	//Action: "InitTool"
	bInitTool			: BOOL;
	nStateA_InitTool	: USINT;	
	
	//Action: "Aspirate"
	bAspirate			: BOOL;
	nStateA_Aspirate	: USINT;
	nQuantity			: DINT;
	nFlow				: DINT;
	
	//Action: "Dispense"
	bDispense			: BOOL;
	nStateA_Dispense	: USINT;

	//Action: "DispensePiezo"
	bDispensePiezo			: BOOL;
	nStateA_DispensePiezo	: USINT;
	nDrops					: UINT;
	bDispensePiezoStart		: BOOL;
	bStroboskopeOn			: BOOL;
	bSetDropsFlag			: BOOL := TRUE;	
	nTestResult				: UDINT;	//wird beim PiezoTest durch InteractResponse Arg1 geschrieben bzw. bei Start des Tests zurückgesetzt
	
	//Action: "MoveDilValve"
	bDilMoveValve			: BOOL;
	nStateA_DilMoveValve	: USINT;
	
	//Action: "SetPressure"
	bSetPress			: BOOL;
	fbSetPress			: FB_SetPressure;
	
	//Action: "SwitchPressure"
	eSwitchPressCtrl	: E_PressCtrl;
	
END_VAR

fbPiezoControl(pFbPiezoRef:= pFbPiezoRef);

IF eCurrentState = E_MachineState.MACHINESTATE_Active THEN
	
	IF bInitTool THEN
		A_InitTool();
		IF nStateA_InitTool >= 80 THEN
			IF nStateA_InitTool >= 99 THEN
				bError := TRUE;
			END_IF
			bInitTool := FALSE;
			nStateA_InitTool := 0;
			M_RemoveListEntry(nSearchValue:= E_Action.ACTION_Init);
		END_IF		
	END_IF

	IF bAspirate THEN
		A_Aspirate();
		IF nStateA_Aspirate >= 80 THEN
			IF nStateA_Aspirate >= 99 THEN
				bError := TRUE;	
			END_IF
			bAspirate := FALSE;
			nStateA_Aspirate := 0;
			M_RemoveListEntry(nSearchValue:= E_Action.ACTION_Aspirate);
		END_IF
	END_IF

	IF bDispense THEN
		A_Dispense();
		IF nStateA_Dispense >= 80 THEN
			IF nStateA_Dispense >= 99 THEN
				bError := TRUE;	
			END_IF
			bDispense := FALSE;
			nStateA_Dispense := 0;
			M_RemoveListEntry(nSearchValue:= E_Action.ACTION_Dispense);
		END_IF
	END_IF
	
	IF bDispensePiezo THEN
		A_DispenseDrops();
		IF nStateA_DispensePiezo >= 80 THEN
			IF nStateA_DispensePiezo >= 99 THEN
				bError := TRUE;			
			END_IF
			bDispensePiezo := FALSE;
			nStateA_DispensePiezo := 0;
			M_RemoveListEntry(nSearchValue:= E_Action.ACTION_DispenseDrops);
		END_IF
	END_IF
	
	IF bDilMoveValve THEN
		A_DilMoveValve();
		IF nStateA_DilMoveValve >= 80 THEN
			IF nStateA_DilMoveValve >= 99 THEN
				bError := TRUE;			
			END_IF
			bDilMoveValve := FALSE;
			nStateA_DilMoveValve := 0;
			M_RemoveListEntry(nSearchValue:= E_Action.ACTION_DilMoveValve);
		END_IF
	END_IF
END_IF

SUPER^();	//FB_MzTool aufrufen

//Prozessdaten aktualisieren
IF pFbPiezoRef > 0 THEN
	stProcessData.n32Data[7] := UDINT_TO_DINT(nTestResult);
	stProcessData.n32Data[8] := BOOL_TO_DINT(pFbPiezoRef^.pToolState^.0);
END_IF

IF pPneuChannelPress > 0 THEN
	stProcessData.n32Data[9] := pPneuChannelPress^.P_nCurrentPressure;
END_IF

stProcessData.n32Data[10] :=	BOOL_TO_DINT(fbPCV.P_bPneuValve);

aObjProcData[nNotifyId] := stProcessData;

ACTION A_Aspirate:
IF pDiluter^.P_bError THEN
	stError.ErrorId := pDiluter^.P_nErrorId;
	stError.POUState := nStateA_Aspirate;
	nStateA_Aspirate := 99;
END_IF

CASE nStateA_Aspirate OF
	0:	//Solenoid mit Startparametern starten und Diluter starten
		MEMSET(ADR(stActionDataSpec),0,SIZEOF(stActionDataSpec));
		stActionDataSpec.eAction := E_Action.ACTION_DilPump;
		stActionDataSpec.aParams[1] := E_DilPumpMode.MODE_Suck;
		stActionDataSpec.aParams[2] := nQuantity; 
		stActionDataSpec.aParams[3] := nFlow;
		
		//fbPCV.M_SwitchPneuValve(FALSE);
		
		stError.ErrorId := pDiluter^.M_ExeAction(stActionDataSpec);
		IF stError.ErrorId > 0 THEN
			stError.POUState := nStateA_Aspirate;
			nStateA_Aspirate := 99;
		ELSE
			rAspFrequSweepTime := DINT_TO_REAL(nQuantity) / DINT_TO_REAL(nFlow) * 1000.0;
			rSweepSteps := rAspFrequSweepTime / 10.0; //10ms per Zyklus
			rFrequStep := (rAspFrequSweepEnd - rAspFrequSweepStart) / rSweepSteps;
			rFrequNew := rAspFrequSweepStart; 
			fbPiezoControl.P_nFrequency := REAL_TO_UINT(rAspFrequSweepStart);
			fbPiezoControl.P_nPulse := nAspiratePulse;
			fbPiezoControl.P_nDrops := 0;
			fbPiezoControl.M_StartStop(TRUE);
			rCurrentSweepStep := 0.0;
			nStateA_Aspirate := 1;
		END_IF
		
	1:	//Warten bis Aspiration fertig
		IF NOT pDiluter^.M_GetActionBusy(E_Action.ACTION_DilPump) THEN
			fbPiezoControl.M_StartStop(FALSE);
			//Originalparameter senden, damit keine Zeit beim DispenseDrops verloren geht
			fbPiezoControl.P_nFrequency := nFrequency;
			fbPiezoControl.P_nPulse := nPulse;
			nStateA_Aspirate := 80;
		ELSE
			//Frequenz anpassen
			rCurrentSweepStep := rCurrentSweepStep + 1.0;
			IF rCurrentSweepStep < rSweepSteps THEN
				rFrequNew := rFrequNew + rFrequStep;
			ELSE
				rFrequNew := rAspFrequSweepEnd;
			END_IF
			fbPiezoControl.P_nFrequency := REAL_TO_UINT(rFrequNew);
		END_IF
		
	70:	//Abbrechen
		MEMSET(ADR(stActionDataSpec),0,SIZEOF(stActionDataSpec));
		stActionDataSpec.eAction := E_Action.ACTION_Stop;
		pDiluter^.M_ExeAction(stActionDataSpec);
		fbPiezoControl.M_StartStop(FALSE);
		nStateA_Aspirate := 71;
		
	71:	//Abbrechen
		IF NOT pDiluter^.P_bBusy THEN
			nStateA_Aspirate := 80;
		END_IF
END_CASE

//Errorhandling
IF nStateA_Aspirate = 99 THEN
	stError.Cmd := E_Action.ACTION_Aspirate;
	stError.POU := E_POU.POU_FB_PiezoPip;
	stError.POUAction := E_POUACT.POUACT_A_Aspirate;
	fbErrorList.M_Add(stError);
END_IF
END_ACTION

ACTION A_DilMoveValve:
stError.POUState := nStateA_DilMoveValve;
IF pDiluter^.P_bError THEN
	stError.ErrorId := pDiluter^.P_nErrorId;
	nStateA_DilMoveValve := 99;
END_IF

IF nStateA_DilMoveValve = 0 THEN
	IF NOT pDiluter^.M_GetActionBusy(E_Action.ACTION_DilMoveValve) THEN
		nStateA_DilMoveValve := 80;
	END_IF
END_IF

//Errorhandling
IF nStateA_DilMoveValve = 99 THEN
	stError.Cmd := E_Action.ACTION_DilMoveValve;
	stError.POU := E_POU.POU_FB_PiezoPip;
	stError.POUAction := E_POUACT.POUACT_A_MoveValve;
	fbErrorList.M_Add(stError);
END_IF
END_ACTION

ACTION A_Dispense:
IF pDiluter^.P_bError THEN
	stError.ErrorId := pDiluter^.P_nErrorId;
	stError.POUState := nStateA_Dispense;
	nStateA_Dispense := 99;
END_IF

CASE nStateA_Dispense OF
	0:	fbPiezoControl.P_nDrops := 0;
		nStateA_Dispense := 1;

	1:	MEMSET(ADR(stActionDataSpec),0,SIZEOF(stActionDataSpec));
		stActionDataSpec.eAction := E_Action.ACTION_DilPump;
		stActionDataSpec.aParams[1] := E_DilPumpMode.MODE_Press;
		stActionDataSpec.aParams[2] := nQuantity; 
		stActionDataSpec.aParams[3] := nFlow;
		
		//fbPCV.M_SwitchPneuValve(FALSE);
		
		stError.ErrorId := pDiluter^.M_ExeAction(stActionDataSpec);
		IF stError.ErrorId > 0 THEN
			stError.POUState := nStateA_Dispense;
			nStateA_Dispense := 99;
		ELSE
			rDispFrequSweepTime := DINT_TO_REAL(nQuantity) / DINT_TO_REAL(nFlow) * 1000.0;
			rSweepSteps := rDispFrequSweepTime / 10.0; //10ms per Zyklus
			rFrequStep := (rDispFrequSweepEnd - rDispFrequSweepStart) / rSweepSteps;
			rFrequNew := rDispFrequSweepStart; 
			fbPiezoControl.P_nFrequency := REAL_TO_UINT(rDispFrequSweepStart);
			fbPiezoControl.P_nPulse := nDispensePulse;
			fbPiezoControl.M_StartStop(TRUE);
			rCurrentSweepStep := 0.0;
			nStateA_Dispense := 2;	
		END_IF
		
	2:	//Warten bis Dispensen fertig
		IF NOT pDiluter^.M_GetActionBusy(E_Action.ACTION_DilPump) THEN
			fbPiezoControl.M_StartStop(FALSE);
			//Originalparameter senden, damit keine Zeit beim DispenseDrops verloren geht
			fbPiezoControl.P_nFrequency := nFrequency;
			fbPiezoControl.P_nPulse := nPulse;			
			nStateA_Dispense := 80;
		ELSE
			//Frequenz anpassen
			rCurrentSweepStep := rCurrentSweepStep + 1.0;
			IF rCurrentSweepStep < rSweepSteps THEN
				rFrequNew := rFrequNew + rFrequStep;
			ELSE
				rFrequNew := rDispFrequSweepEnd;
			END_IF
			fbPiezoControl.P_nFrequency := REAL_TO_UINT(rFrequNew);
		END_IF
		
	70:	//Abbrechen
		MEMSET(ADR(stActionDataSpec),0,SIZEOF(stActionDataSpec));
		stActionDataSpec.eAction := E_Action.ACTION_Stop;
		pDiluter^.M_ExeAction(stActionDataSpec);
		fbPiezoControl.M_StartStop(FALSE);		
		nStateA_Dispense := 71;
		
	71:	
		IF NOT pDiluter^.P_bBusy THEN
			nStateA_Dispense := 80;
		END_IF
		
END_CASE

//Errorhandling
IF nStateA_Dispense = 99 THEN
	stError.Cmd := E_Action.ACTION_Dispense;
	stError.POU := E_POU.POU_FB_PiezoPip;
	stError.POUAction := E_POUACT.POUACT_A_Dispense;
	fbErrorList.M_Add(stError);
END_IF
END_ACTION

ACTION A_DispenseDrops:
CASE nStateA_DispensePiezo OF
	0:	//Wenn Diluter nicht auf Bypass, dann auf Bypass stellen
		IF pDiluter^.P_nCurValvePos <> 3 THEN
			MEMSET(ADR(stActionDataSpec),0,SIZEOF(stActionDataSpec));
			stActionDataSpec.eAction := E_Action.ACTION_DilMoveValve;
			stActionDataSpec.aParams[1] := 3;
			stError.ErrorId := pDiluter^.M_ExeAction(stActionDataSpec);
			IF stError.ErrorId > 0 THEN
				stError.POUState := nStateA_DispensePiezo;
				nStateA_DispensePiezo := 99;
			ELSE
				nStateA_DispensePiezo := 1;
			END_IF
		ELSE
			nStateA_DispensePiezo := 1;
		END_IF
		
		//Druck auf PCV geben
		fbPCV.M_SwitchPneuValve(TRUE);
	
	1:	//Warten, bis Diluter fertig und Drops übertragen
		IF pDiluter^.P_bError THEN
			stError.ErrorId := pDiluter^.P_nErrorId;	
			stError.POUState := nStateA_DispensePiezo;
			nStateA_DispensePiezo := 99;
		ELSE
			//Dispensen erst starten, nachdem alle Parameter gesendet
			IF (NOT pDiluter^.M_GetActionBusy(E_Action.ACTION_DilMoveValve)) AND NOT (fbPiezoControl.P_bIsSending) THEN
				fbPiezoControl.M_StartStop(bDispensePiezoStart); //Piezo starten
				nStateA_DispensePiezo := 2;
			END_IF
		END_IF
		
	2: 	//Warten bis Piezo fertig
		IF NOT fbPiezoControl.bBusy THEN
			nStateA_DispensePiezo := 80;	
		END_IF
		
		IF fbPiezoControl.bError THEN
			stError.ErrorId := fbPiezoControl.nErrorId;
			stError.POUState := nStateA_DispensePiezo;
			nStateA_DispensePiezo := 99;
		END_IF
		
	70:	//Abbrechen
		fbPiezoControl.M_StartStop(FALSE);
		nStateA_DispensePiezo := 80;		
 END_CASE

//Errorhandling
IF nStateA_DispensePiezo = 99 THEN
	stError.Cmd := E_Action.ACTION_DispenseDrops;
	stError.POU := E_POU.POU_FB_PiezoPip;
	stError.POUAction := E_POUACT.POUACT_A_DispensePiezo;
	fbErrorList.M_Add(stError);
END_IF
END_ACTION

ACTION A_InitTool:
IF nStateA_InitTool = 0 THEN
	pFbPiezoRef^.P_eDispenserMode := E_DispenserMode.MODE_Solenoid;
	fbPiezoControl.M_Init();
	bInitToolOk := TRUE;
	nStateA_InitTool := 80;
END_IF
END_ACTION

ACTION A_Reset:
//Ist noch eine Aktion aktiv?
IF nStateA_ResetSpec = 0 THEN 
	IF bAspirate THEN
		bAspirate := FALSE;
		nStateA_Aspirate := 0;
	END_IF

	IF bDispense THEN
		bDispense := FALSE;
		nStateA_Dispense := 0;
	END_IF

	IF bDispensePiezo THEN
		bDispensePiezo := FALSE;
		nStateA_DispensePiezo := 0;
	END_IF
	
	IF bSetPress THEN
		bSetPress := FALSE;
		fbSetPress(bExecute:= FALSE, pPneuChannelRef:= pPneuChannelPress);
	END_IF

	nStateA_ResetSpec := 80;
END_IF

SUPER^.A_Reset();
END_ACTION

ACTION A_Stop:
IF nStateA_Stop = 0 THEN

	IF bSetPress THEN
		fbSetPress(bExecute:= FALSE, pPneuChannelRef:= pPneuChannelPress);
	END_IF
	
	IF bAspirate AND nStateA_Aspirate < 70 THEN
		nStateA_Aspirate := 70;
	END_IF

	IF bDispense AND nStateA_Dispense < 70 THEN
		nStateA_Dispense := 70;
	END_IF

	IF bDispensePiezo AND nStateA_DispensePiezo < 70 THEN
		nStateA_DispensePiezo := 70;
	END_IF
	
	nStateA_Stop := 1;
END_IF

SUPER^.A_Stop();
END_ACTION

METHOD FB_init : BOOL
VAR_INPUT
	bInitRetains : BOOL; // if TRUE, the retain variables are initialized (warm start / cold start)
	bInCopyCode : BOOL;  // if TRUE, the instance afterwards gets moved into the copy code (online change)
END_VAR
eObjectType := E_ObjectType.OBJECTTYPE_SolenoidPip;
eObjectGroup := E_ObjectGroup.OBJECTGROUP_MzTool OR E_ObjectGroup.OBJECTGROUP_Device;
END_METHOD

METHOD M_AddChild : ERRORID
VAR_INPUT
	pObject : POINTER TO FB_Object;
	nSlotNr	: UINT;
	nIndex 	: INT;
END_VAR
//Kann keine Objekte aufnehmen
M_AddChild := E_ErrorIdObjMgmt.ERRORID_ObjectCanNotTakeChilds;
END_METHOD

METHOD M_CancelAction
VAR_INPUT
	eAction : E_Action;
END_VAR
CASE eAction OF
	E_Action.ACTION_Aspirate:
		IF bAspirate AND nStateA_Aspirate < 70 THEN
			nStateA_Aspirate := 70;
		END_IF
	E_Action.ACTION_Dispense:
		IF bDispense AND nStateA_Dispense < 70 THEN
			nStateA_Dispense := 70;
		END_IF
	E_Action.ACTION_DispenseDrops:
		IF bDispensePiezo AND nStateA_DispensePiezo < 70 THEN
			nStateA_DispensePiezo := 70;
		END_IF
	E_Action.ACTION_SetPressure:
		IF bSetPress THEN
			fbSetPress(bExecute:= FALSE, pPneuChannelRef:= pPneuChannelPress);
		END_IF
ELSE
	SUPER^.M_CancelAction(eAction);
END_CASE
END_METHOD

METHOD M_CheckAction : ERRORID
VAR_INPUT
	refActionData 	: REFERENCE TO ST_ActionData;
	pCorrelObject	: POINTER TO FB_Object;
END_VAR

VAR
	pTarget : POINTER TO FB_TargetBase;
	pRack	: POINTER TO FB_Rack;
	pSlot	: POINTER TO FB_PieceSlot;		
END_VAR
CASE refActionData.eAction OF
	E_Action.ACTION_Dispense, //BasicAction für ActionOnArray
	E_Action.ACTION_Aspirate, //BasicAction für ActionOnArray
	E_Action.ACTION_DispenseDrops, //BasicAction für ActionOnArray
	E_Action.ACTION_DispenseTest,
	E_Action.ACTION_GetPipSample,
	E_Action.ACTION_MeasureTool,
	E_Action.ACTION_TeachTarget:
		RETURN;
	E_Action.ACTION_WashTool:
		//Washmode checken
		IF refActionData.aParams[2] = E_WashMode.MODE_WashInside THEN
			M_CheckAction := M_CheckBottles();
		ELSIF refActionData.aParams[2] = E_WashMode.MODE_WashOutside THEN
			;
		ELSIF refActionData.aParams[2] = E_WashMode.MODE_WashInOutside THEN
			M_CheckAction := M_CheckBottles();
		ELSIF refActionData.aParams[2] = E_WashMode.MODE_DryOutside THEN
			;
		ELSE
			M_CheckAction := E_ErrorIdCmd.ERRORID_InvalidWashMode;	
		END_IF
	E_Action.ACTION_InsertTool:
		//SolenoidPip darf nur in offene Vials oder Fliptubes eintauchen
		//-> Target muss also ein VialRack sein (Reaktor nicht möglich, da Pip nicht von der Tiefe hinein passt)
		pTarget := pCorrelObject;
		IF pTarget > 0 THEN
			IF (pTarget^.P_eObjectGroup AND E_ObjectGroup.OBJECTGROUP_Rack) = E_ObjectGroup.OBJECTGROUP_Rack THEN
				pRack := pTarget;
				pSlot := pRack^.M_GetSlot(DINT_TO_UINT(refActionData.aParams[2]));
				IF pSlot > 0 THEN
					IF pSlot^.P_pPiece = 0 THEN
						M_CheckAction := E_ErrorIdCmd.ERRORID_NoPieceInSlot;
						RETURN;
					ELSIF NOT (pSlot^.P_pPiece^.P_eObjectType = E_ObjectType.OBJECTTYPE_Vial OR pSlot^.P_pPiece^.P_eObjectType = E_ObjectType.OBJECTTYPE_FlipTube) THEN
						M_CheckAction := E_ErrorIdCmd.ERRORID_InvalidPieceType;
					END_IF
				ELSE
					M_CheckAction := E_ErrorIdCmd.ERRORID_InvalidTargetSlot;
					RETURN;
				END_IF	
			ELSE
				M_CheckAction := E_ErrorIdCmd.ERRORID_UnsuitableTarget;	
			END_IF
		ELSE
			M_CheckAction := E_ErrorIdCmd.ERRORID_UnsuitableTarget;	
		END_IF		
ELSE
	M_CheckAction := SUPER^.M_CheckAction(refActionData, pCorrelObject);
END_CASE
END_METHOD

METHOD M_CheckBottles : ERRORID
VAR_INPUT
END_VAR
IF pDiluter > 0 THEN
	M_CheckBottles := 0;
END_IF
END_METHOD

METHOD M_CheckProps : ERRORID
VAR_INPUT
END_VAR
M_CheckProps := SUPER^.M_CheckProps();
IF M_CheckProps > 0 THEN
	RETURN;
END_IF
//Konfigurierte Properties checken
//zugeordneter Diuter
IF fbObjectDirectory.M_GetObjType(nDiluterObjId) <> E_ObjectType.OBJECTTYPE_Diluter THEN
	M_CheckProps := E_ErrorIdObjMgmt.ERRORID_InvalidDiluterObjId; //Error
	RETURN;
ELSE
	pDiluter := fbObjectDirectory.M_GetObjPointer(nDiluterObjId);
END_IF
END_METHOD

METHOD M_ClearAllProps
VAR_INPUT
	bIgnoreParent : BOOL; //Es wird das gesamte OD gelöscht. -> Zeiger auf Parent nicht mehr gültig!
END_VAR
pPneuChannelPress := 0;
SUPER^.M_ClearAllProps(bIgnoreParent);
END_METHOD

METHOD M_ExeAction : ERRORID
VAR_INPUT
	refActionData : REFERENCE TO ST_ActionData;	
END_VAR
IF NOT (eCurrentState = E_MachineState.MACHINESTATE_Idle OR
	eCurrentState = E_MachineState.MACHINESTATE_Active OR
	eCurrentState = E_MachineState.MACHINESTATE_Ready) THEN
	M_ExeAction := E_ErrorIdCmd.ERRORID_InvalidState;
	RETURN;
END_IF

CASE refActionData.eAction OF
	
	E_Action.ACTION_Init:
		IF NOT bInitAxis AND NOT bInitTool THEN
			bInitAxis := TRUE;
			bInitTool := TRUE;
			fbList.A_AddHeadValue( hList := hList, putValue := E_Action.ACTION_Init);	//InitBase
			fbList.A_AddHeadValue( hList := hList, putValue := E_Action.ACTION_Init);	//InitSpec
		ELSE
			RETURN;
		END_IF		
	
	E_Action.ACTION_Aspirate:
		IF NOT bAspirate THEN
			M_ExeAction := pDiluter^.M_CheckBottles(0); //Checken, ob Bottles OK
			IF M_ExeAction > 0 THEN
				RETURN;
			END_IF
			nQuantity := refActionData.aParams[1];
			nFlow := refActionData.aParams[2];
			fbList.A_AddHeadValue( hList := hList, putValue := E_Action.ACTION_Aspirate);
			bAspirate := TRUE;
		END_IF
		
	E_Action.ACTION_Dispense:
		IF NOT bDispense THEN
			M_ExeAction := pDiluter^.M_CheckBottles(0); //Checken, ob Bottles OK
			IF M_ExeAction > 0 THEN
				RETURN;
			END_IF
			nQuantity := refActionData.aParams[1];
			nFlow := refActionData.aParams[2];
			fbList.A_AddHeadValue( hList := hList, putValue := E_Action.ACTION_Dispense);
			bDispense := TRUE;
		END_IF
		
	E_Action.ACTION_DispenseDrops:
		bDispensePiezoStart := DINT_TO_BOOL(refActionData.aParams[2]);
		IF NOT bDispensePiezo AND bDispensePiezoStart THEN
			fbPiezoControl.P_nFrequency := nFrequency;
			fbPiezoControl.P_nPulse := nPulse;
			fbPiezoControl.P_nDrops := nDrops := DINT_TO_UINT(refActionData.aParams[1]);
			fbPiezoControl.P_bStroboscope := DINT_TO_BOOL(refActionData.aParams[3]);
			fbList.A_AddHeadValue(hList := hList, putValue := E_Action.ACTION_DispenseDrops);
			bDispensePiezo := TRUE;
		ELSE
			fbPiezoControl.M_StartStop(bDispensePiezoStart); //Stoppen
		END_IF
		
	E_Action.ACTION_DilMoveValve:
		//Darf nur ausgeführt werden, wenn kein Dispensen aktiv ist
		IF NOT (bAspirate OR bDispense OR bDispensePiezo OR bDilMoveValve) THEN
			M_ExeAction := pDiluter^.M_ExeAction(refActionData);
			IF M_ExeAction > 0 THEN
				RETURN;
			END_IF
			fbList.A_AddHeadValue(hList := hList, putValue := E_Action.ACTION_DilMoveValve);
			bDilMoveValve := TRUE;
		END_IF
		
	E_Action.ACTION_MoveX,E_Action.ACTION_MoveY,E_Action.ACTION_MoveXY:
		IF pZAxisRef^.stInput.nToolState.1 THEN	//ZSensor ist montiert
			M_ExeAction := ERRORID_PipMoveWithZSensor;  //Error
			RETURN;
		ELSE
			M_ExeAction := SUPER^.M_ExeAction(refActionData);
			RETURN;
		END_IF

	E_Action.ACTION_MoveZ:
		IF pZAxisRef^.stInput.nToolState.1 THEN //ZSensor ist montiert
			eMoveModeZ := DINT_TO_USINT(refActionData.aParams[1]);
			IF NOT(eMoveModeZ = E_MoveMode.MODE_Free OR eMoveModeZ = E_MoveMode.MODE_Home) THEN
				M_ExeAction := ERRORID_PipMoveWithZSensor;  //Error
				RETURN;
			END_IF
			M_ExeAction := SUPER^.M_ExeAction(refActionData);
			RETURN;			
		ELSE
			M_ExeAction := SUPER^.M_ExeAction(refActionData);
			RETURN;
		END_IF
		
	E_Action.ACTION_SetPressure:
		fbSetPress(bExecute:= FALSE, pPneuChannelRef:= pPneuChannelPress); //eventueller Fehler wird auch zurückgesetzt
		fbSetPress.bAwait := DINT_TO_BOOL(refActionData.aParams[1]);
		fbSetPress.nValue := DINT_TO_INT(refActionData.aParams[2]);
		fbSetPress.nTolerancePlus := DINT_TO_INT(refActionData.aParams[3]);
		fbSetPress.nToleranceMinus := DINT_TO_INT(refActionData.aParams[4]);
		fbSetPress.tTimeout := DINT_TO_TIME(refActionData.aParams[5]);
		
		fbSetPress(bExecute:= TRUE,	pPneuChannelRef:= pPneuChannelPress,nErrorId=> M_ExeAction);
		IF fbSetPress.bError THEN
			RETURN;
		END_IF
		
		IF NOT bSetPress AND fbSetPress.bBusy THEN
			bSetPress := TRUE;
			fbList.A_AddHeadValue(hList := hList, putValue := E_Action.ACTION_SetPressure);
		ELSE
			RETURN;	
		END_IF
		
	E_Action.ACTION_SwitchPressure:
		eSwitchPressCtrl := DINT_TO_USINT(refActionData.aParams[1]);
		IF eSwitchPressCtrl = E_PressCtrl.PRESSCTRL_PressOn THEN
			fbPCV.M_SwitchPneuValve(TRUE);
		ELSIF eSwitchPressCtrl = E_PressCtrl.PRESSCTRL_Off THEN
			fbPCV.M_SwitchPneuValve(FALSE);
		ELSE
			M_ExeAction := E_ErrorIdCmd.ERRORID_InvalidCtrl;
			RETURN;		
		END_IF
	ELSE
		M_ExeAction := SUPER^.M_ExeAction(refActionData);
		RETURN;
END_CASE
bBusy := TRUE;
eCurrentState := E_MachineState.MACHINESTATE_Active;
END_METHOD

METHOD M_GetAllProps : ERRORID
VAR_INPUT
	refCmdData : REFERENCE TO  ST_CmdData;
END_VAR
//BaseProperties lesen
SUPER^.M_GetAllProps(refCmdData);
nCurrentPropIndex := nCurrentPropIndex + 1;
refCmdData.n32Data[nCurrentPropIndex] := P_nObjIdDiluter;
nCurrentPropIndex := nCurrentPropIndex + 1;
IF pPneuChannelPress > 0 THEN
	refCmdData.n32Data[nCurrentPropIndex] := pPneuChannelPress^.nChannel;
ELSE
	refCmdData.n32Data[nCurrentPropIndex] := 0;
END_IF
nCurrentPropIndex := nCurrentPropIndex + 1;
refCmdData.n32Data[nCurrentPropIndex] := nFrequency;
nCurrentPropIndex := nCurrentPropIndex + 1;
refCmdData.n32Data[nCurrentPropIndex] := nPulse;
nCurrentPropIndex := nCurrentPropIndex + 1;
refCmdData.n32Data[nCurrentPropIndex] := fbPiezoControl.P_nHoldVoltage;
nCurrentPropIndex := nCurrentPropIndex + 1;
refCmdData.n32Data[nCurrentPropIndex] := fbPiezoControl.P_nPrePeakTime;
nCurrentPropIndex := nCurrentPropIndex + 1;
refCmdData.n32Data[nCurrentPropIndex] := REAL_TO_DINT(rAspFrequSweepStart);
nCurrentPropIndex := nCurrentPropIndex + 1;
refCmdData.n32Data[nCurrentPropIndex] := REAL_TO_DINT(rAspFrequSweepEnd);
nCurrentPropIndex := nCurrentPropIndex + 1;
refCmdData.n32Data[nCurrentPropIndex] := REAL_TO_DINT(rAspFrequSweepTime);
nCurrentPropIndex := nCurrentPropIndex + 1;
refCmdData.n32Data[nCurrentPropIndex] := nAspiratePulse;
nCurrentPropIndex := nCurrentPropIndex + 1;
refCmdData.n32Data[nCurrentPropIndex] := REAL_TO_DINT(rDispFrequSweepStart);
nCurrentPropIndex := nCurrentPropIndex + 1;
refCmdData.n32Data[nCurrentPropIndex] := REAL_TO_DINT(rDispFrequSweepEnd);
nCurrentPropIndex := nCurrentPropIndex + 1;
refCmdData.n32Data[nCurrentPropIndex] := REAL_TO_DINT(rDispFrequSweepTime);
nCurrentPropIndex := nCurrentPropIndex + 1;
refCmdData.n32Data[nCurrentPropIndex] := nDispensePulse;
nCurrentPropIndex := nCurrentPropIndex + 1;
refCmdData.n32Data[nCurrentPropIndex] := nDrypadArea;
nCurrentPropIndex := nCurrentPropIndex + 1;
refCmdData.n32Data[nCurrentPropIndex] := TIME_TO_DINT(tDryTime);
END_METHOD

METHOD M_SetAllProps : ERRORID
VAR_INPUT
	refCmdData : REFERENCE TO  ST_CmdData;
END_VAR

VAR
	pSinglePiezoHolder 	: POINTER TO FB_SingelPiezoHolder;
	pTwinPiezoHolder 	:  POINTER TO FB_TwinPiezoHolder;
	nPneuChannel 		: USINT;
END_VAR
M_SetAllProps := SUPER^.M_SetAllProps(refCmdData);

IF M_SetAllProps > 0 THEN
	RETURN;
END_IF

IF pParentMzTool^.P_eObjectType = E_ObjectType.OBJECTTYPE_SinglePiezoHolder THEN
	pSinglePiezoHolder := pParentMzTool;
	pFbPiezoRef := pSinglePiezoHolder^.M_GetPiezoRef(pParentSlot);	
ELSIF pParentMzTool^.P_eObjectType = E_ObjectType.OBJECTTYPE_TwinPiezoHolder THEN
	pTwinPiezoHolder := pParentMzTool;
	pFbPiezoRef := pTwinPiezoHolder^.M_GetPiezoRef(pParentSlot);
ELSE
	M_SetAllProps := E_ErrorIdObjMgmt.ERRORID_InvalidParentMzTool;
	RETURN;
END_IF

IF pFbPiezoRef = 0 THEN
	M_SetAllProps := E_ErrorIdObjMgmt.ERRORID_InvalidPiezoRef;
	RETURN;
END_IF

fbPiezoControl(pFbPiezoRef:= pFbPiezoRef);	//Setzt den Zeiger "pFbPiezoRef" innerhalb von fbMultiZPiezo

//Diluter
nCurrentPropIndex := nCurrentPropIndex + 1;
nSpecPropIndex := nCurrentPropIndex;
nDiluterObjId :=  DINT_TO_UINT(refCmdData.n32Data[nCurrentPropIndex]);
IF fbObjectDirectory.M_GetObjType(nDiluterObjId) = E_ObjectType.OBJECTTYPE_Diluter THEN
	pDiluter := fbObjectDirectory.M_GetObjPointer(nDiluterObjId);
ELSE
	M_SetAllProps := E_ErrorIdObjMgmt.ERRORID_InvalidDiluterObjId;
	RETURN;
END_IF

//PneuChannel
nCurrentPropIndex := nCurrentPropIndex + 1;
nPneuChannel := DINT_TO_USINT(refCmdData.n32Data[nCurrentPropIndex]);	//PneuChannel Druck
IF NOT (nPneuChannel > 0 AND nPneuChannel <= cNoOfPneuChannels) THEN
	M_SetAllProps := E_ErrorIdObjMgmt.ERRORID_InvalidPneuChannel;
	RETURN;	
END_IF
pPneuChannelPress := ADR(aFbPneuChannel[nPneuChannel]);

//Frequenz
nCurrentPropIndex := nCurrentPropIndex + 1;
M_SetAllProps := M_SetFrequency(refCmdData.n32Data[nCurrentPropIndex], FALSE);
IF M_SetAllProps > 0 THEN
	RETURN;
END_IF

//Plusbreite
nCurrentPropIndex := nCurrentPropIndex + 1;
M_SetAllProps := M_SetPulse(refCmdData.n32Data[nCurrentPropIndex], FALSE);
IF M_SetAllProps > 0 THEN
	RETURN;
END_IF

//Spannung (HoldVoltage) in mV
nCurrentPropIndex := nCurrentPropIndex + 1;
M_SetAllProps := M_SetVoltage(refCmdData.n32Data[nCurrentPropIndex], FALSE);
IF M_SetAllProps > 0 THEN
	RETURN;
END_IF

//PrePeakTime
nCurrentPropIndex := nCurrentPropIndex + 1;
IF NOT (refCmdData.n32Data[nCurrentPropIndex] >= 100 AND refCmdData.n32Data[nCurrentPropIndex] <= 350) THEN
	M_SetAllProps := E_ErrorIdObjMgmt.ERRORID_InvalidPrePeakTime;
	RETURN;
END_IF
fbPiezoControl.P_nPrePeakTime := DINT_TO_UINT(refCmdData.n32Data[nCurrentPropIndex]);

//FrequenzSweep Anfangsfrequenz - Aspirieren
nCurrentPropIndex := nCurrentPropIndex + 1;
IF NOT (refCmdData.n32Data[nCurrentPropIndex] >= 30 AND refCmdData.n32Data[nCurrentPropIndex] <= 500) THEN
	M_SetAllProps := E_ErrorIdObjMgmt.ERRORID_InvalidFrequency;
	RETURN;
END_IF
rAspFrequSweepStart := DINT_TO_REAL(refCmdData.n32Data[nCurrentPropIndex]);

//FrequenzSweep Endfrequenz - Aspirieren
nCurrentPropIndex := nCurrentPropIndex + 1;
IF NOT (refCmdData.n32Data[nCurrentPropIndex] >= 30 AND refCmdData.n32Data[nCurrentPropIndex] <= 500) THEN
	M_SetAllProps := E_ErrorIdObjMgmt.ERRORID_InvalidFrequency;
	RETURN;
END_IF
rAspFrequSweepEnd := DINT_TO_REAL(refCmdData.n32Data[nCurrentPropIndex]);

//FrequenzSweep Zeit - Aspirieren
nCurrentPropIndex := nCurrentPropIndex + 1;
rAspFrequSweepTime := DINT_TO_REAL(refCmdData.n32Data[nCurrentPropIndex]);

 //Pulsbreite - Aspirieren
nCurrentPropIndex := nCurrentPropIndex + 1;
IF NOT (refCmdData.n32Data[nCurrentPropIndex] >= 400 AND refCmdData.n32Data[nCurrentPropIndex] <= 10000) THEN
	M_SetAllProps := E_ErrorIdObjMgmt.ERRORID_InvalidPulseWidth;
	RETURN;
END_IF
nAspiratePulse := DINT_TO_UINT(refCmdData.n32Data[nCurrentPropIndex]);

//FrequenzSweep Anfangsfrequenz - Dispensen
nCurrentPropIndex := nCurrentPropIndex + 1;
IF NOT (refCmdData.n32Data[nCurrentPropIndex] >= 30 AND refCmdData.n32Data[nCurrentPropIndex] <= 500) THEN
	M_SetAllProps := E_ErrorIdObjMgmt.ERRORID_InvalidFrequency;
	RETURN;
END_IF
rDispFrequSweepStart := DINT_TO_REAL(refCmdData.n32Data[nCurrentPropIndex]);

//FrequenzSweep Endfrequenz - Dispensen
nCurrentPropIndex := nCurrentPropIndex + 1;
IF NOT (refCmdData.n32Data[nCurrentPropIndex] >= 30 AND refCmdData.n32Data[nCurrentPropIndex] <= 500) THEN
	M_SetAllProps := E_ErrorIdObjMgmt.ERRORID_InvalidFrequency;
	RETURN;
END_IF
rDispFrequSweepEnd := DINT_TO_REAL(refCmdData.n32Data[nCurrentPropIndex]);

//FrequenzSweep Zeit - Dispensen
nCurrentPropIndex := nCurrentPropIndex + 1;
rDispFrequSweepTime := DINT_TO_REAL(refCmdData.n32Data[nCurrentPropIndex]);

 //Pulsbreite - Dispensen
nCurrentPropIndex := nCurrentPropIndex + 1;
IF NOT (refCmdData.n32Data[nCurrentPropIndex] >= 400 AND refCmdData.n32Data[nCurrentPropIndex] <= 10000) THEN
	M_SetAllProps := E_ErrorIdObjMgmt.ERRORID_InvalidPulseWidth;
	RETURN;
END_IF
nDispensePulse := DINT_TO_UINT(refCmdData.n32Data[nCurrentPropIndex]);

//DrypadArea
nCurrentPropIndex := nCurrentPropIndex + 1;
nDrypadArea := DINT_TO_USINT(refCmdData.n32Data[nCurrentPropIndex]);
IF NOT (nDrypadArea > 0 AND nDrypadArea < 3) THEN
	M_SetAllProps := E_ErrorIdObjMgmt.ERRORID_InvalidDrypadArea;
	RETURN;
END_IF

//DryTime
nCurrentPropIndex := nCurrentPropIndex + 1;
tDryTime := DINT_TO_TIME(refCmdData.n32Data[nCurrentPropIndex]);

nNoOfProps := nCurrentPropIndex + 1;
END_METHOD

METHOD M_SetFrequency : ERRORID
VAR_INPUT
	nValue 				: DINT;
	bSetObjectChange 	: BOOL;
END_VAR
IF nValue >= 30 AND nValue < 500 THEN
	fbPiezoControl.P_nFrequency := nFrequency := DINT_TO_UINT(nValue);
	IF bSetObjectChange THEN
		fbObjectDirectory.M_SetObjChange(nObjectId);
	END_IF	
ELSE
	M_SetFrequency := E_ErrorIdObjMgmt.ERRORID_InvalidFrequency;
END_IF
END_METHOD

METHOD M_SetPrintParams : ST_MethResult
VAR_INPUT
	eType 		: E_PrintParamType;
	nNumerator	: USINT;
	nValue		: DINT;
END_VAR
IF nNumerator <> 1 THEN
	M_SetPrintParams.bError := TRUE;
	M_SetPrintParams.nErrorId := E_ErrorIdCmd.ERRORID_InvalidPrintParamNumerator;
	RETURN;
END_IF

CASE eType OF
	E_PrintParamType.Frequency:
		M_SetPrintParams.nErrorId := M_SetFrequency(nValue, TRUE);
	E_PrintParamType.Pulse:
		M_SetPrintParams.nErrorId := M_SetPulse(nValue, TRUE);
	E_PrintParamType.Voltage:
		M_SetPrintParams.nErrorId := M_SetVoltage(nValue, TRUE);
ELSE
	M_SetPrintParams.bError := TRUE;
	M_SetPrintParams.nErrorId := E_ErrorIdCmd.ERRORID_InvalidPrintParamType;
END_CASE

IF M_SetPrintParams.nErrorId > 0 THEN
	M_SetPrintParams.bError := TRUE;
ELSE
	fbObjectDirectory.M_SetObjChange(nObjectId);
END_IF
END_METHOD

METHOD M_SetPulse : ERRORID
VAR_INPUT
	nValue 				: DINT;
	bSetObjectChange 	: BOOL;
END_VAR
IF nValue > 400 AND nValue < 10000 THEN
	fbPiezoControl.P_nPulse := nPulse := DINT_TO_UINT(nValue);
	IF bSetObjectChange THEN
		fbObjectDirectory.M_SetObjChange(nObjectId);
	END_IF	
ELSE
	M_SetPulse := E_ErrorIdObjMgmt.ERRORID_InvalidPulseWidth;
END_IF
END_METHOD

METHOD M_SetSingleProp : ERRORID
VAR_INPUT
	refCmdData : REFERENCE TO  ST_CmdData;
END_VAR
VAR
	rAspDispTime	: REAL;
	nPneuChannel 	: USINT;
END_VAR
IF nSpecPropIndex = refCmdData.aHeader[1] THEN
	//Diluter Id sollte nicht einzeln geändert werden können!
	M_SetSingleProp := E_ErrorIdCmd.ERRORID_InvalidProperty;

ELSIF (nSpecPropIndex + 1) = refCmdData.aHeader[1] THEN	//PneuChannel
	nPneuChannel := DINT_TO_USINT(refCmdData.n32Data[0]);	//PneuChannel Druck
	IF NOT (nPneuChannel > 0 AND nPneuChannel <= cNoOfPneuChannels) THEN
		M_SetSingleProp := E_ErrorIdObjMgmt.ERRORID_InvalidPneuChannel;
		RETURN;	
	END_IF
	pPneuChannelPress := ADR(aFbPneuChannel[nPneuChannel]);	

ELSIF (nSpecPropIndex + 2) = refCmdData.aHeader[1] THEN	//Frequenz
	M_SetSingleProp := M_SetFrequency(refCmdData.n32Data[0], FALSE);
	
ELSIF (nSpecPropIndex + 3) = refCmdData.aHeader[1] THEN //Pulsbreite
	M_SetSingleProp := M_SetPulse(refCmdData.n32Data[0], FALSE);
	
ELSIF (nSpecPropIndex + 4) = refCmdData.aHeader[1] THEN	//Spannung (HoldVoltage)
	M_SetSingleProp := M_SetVoltage(refCmdData.n32Data[0], FALSE);
	
ELSIF (nSpecPropIndex + 5) = refCmdData.aHeader[1] THEN	//PrePeakTime
	IF NOT (refCmdData.n32Data[0] >= 100 AND refCmdData.n32Data[0] <= 350) THEN
		M_SetSingleProp := E_ErrorIdObjMgmt.ERRORID_InvalidPrePeakTime;;
		RETURN;		
	END_IF
	fbPiezoControl.P_nPrePeakTime := DINT_TO_UINT(refCmdData.n32Data[0]);
	
ELSIF (nSpecPropIndex + 6) = refCmdData.aHeader[1] THEN
	IF NOT (refCmdData.n32Data[0] >= 30 AND refCmdData.n32Data[0] <= 500) THEN //FrequenzSweep Anfangsfrequenz - Aspirieren
		M_SetSingleProp := E_ErrorIdObjMgmt.ERRORID_InvalidFrequency;
		RETURN;
	END_IF
	rAspFrequSweepStart := DINT_TO_REAL(refCmdData.n32Data[0]);
	
ELSIF (nSpecPropIndex + 7) = refCmdData.aHeader[1] THEN
	IF NOT (refCmdData.n32Data[0] >= 30 AND refCmdData.n32Data[0] <= 500) THEN //FrequenzSweep Endfrequenz - Aspirieren
		M_SetSingleProp := E_ErrorIdObjMgmt.ERRORID_InvalidFrequency;
		RETURN;
	END_IF
	rAspFrequSweepEnd := DINT_TO_REAL(refCmdData.n32Data[0]);
	
ELSIF (nSpecPropIndex + 8) = refCmdData.aHeader[1] THEN //FrequenzSweep Zeit - Aspirieren
	rAspFrequSweepTime := DINT_TO_REAL(refCmdData.n32Data[0]);
	
ELSIF (nSpecPropIndex + 9) = refCmdData.aHeader[1] THEN
	IF NOT (refCmdData.n32Data[0] >= 400 AND refCmdData.n32Data[0] <= 10000) THEN //Pulsbreite - Aspirieren
		M_SetSingleProp := E_ErrorIdObjMgmt.ERRORID_InvalidPulseWidth;
		RETURN;
	END_IF
	//Falls entsprechende Aktion aktiv, dann gleich zur Hardware senden	
	nAspiratePulse := DINT_TO_UINT(refCmdData.n32Data[0]);
	
ELSIF (nSpecPropIndex + 10) = refCmdData.aHeader[1] THEN
	IF NOT (refCmdData.n32Data[0] >= 30 AND refCmdData.n32Data[0] <= 500) THEN //FrequenzSweep Anfangsfrequenz - Dispensen
		M_SetSingleProp := E_ErrorIdObjMgmt.ERRORID_InvalidFrequency;
		RETURN;
	END_IF
	rDispFrequSweepStart := DINT_TO_REAL(refCmdData.n32Data[0]);
	
ELSIF (nSpecPropIndex + 11) = refCmdData.aHeader[1] THEN
	IF NOT (refCmdData.n32Data[0] >= 30 AND refCmdData.n32Data[0] <= 500) THEN //FrequenzSweep Endfrequenz - Dispensen
		M_SetSingleProp := E_ErrorIdObjMgmt.ERRORID_InvalidFrequency;
		RETURN;
	END_IF
	rDispFrequSweepEnd := DINT_TO_REAL(refCmdData.n32Data[0]);

ELSIF (nSpecPropIndex + 12) = refCmdData.aHeader[1] THEN //FrequenzSweep Zeit - Dispensen
	rDispFrequSweepTime := DINT_TO_REAL(refCmdData.n32Data[0]);
	
ELSIF (nSpecPropIndex + 13) = refCmdData.aHeader[1] THEN
	IF NOT (refCmdData.n32Data[0] >= 400 AND refCmdData.n32Data[0] <= 10000) THEN //Pulsbreite - Dispensen
		M_SetSingleProp := E_ErrorIdObjMgmt.ERRORID_InvalidPulseWidth;
		RETURN;
	END_IF
	nDispensePulse := DINT_TO_UINT(refCmdData.n32Data[0]);
	
ELSIF (nSpecPropIndex + 14) = refCmdData.aHeader[1] THEN //DryTime
	tDryTime := DINT_TO_TIME(refCmdData.n32Data[0]);
ELSE
	M_SetSingleProp := SUPER^.M_SetSingleProp(refCmdData);
END_IF
END_METHOD

METHOD M_SetVoltage : ERRORID
VAR_INPUT
	nValue 				: DINT;
	bSetObjectChange 	: BOOL;
END_VAR
IF nValue > 1500 AND nValue < 4500 THEN
	fbPiezoControl.P_nHoldVoltage := DINT_TO_UINT(nValue);
	IF bSetObjectChange THEN
		fbObjectDirectory.M_SetObjChange(nObjectId);
	END_IF	
ELSE
	M_SetVoltage := E_ErrorIdObjMgmt.ERRORID_InvalidVoltage;
END_IF
END_METHOD

METHOD M_StartUniDispense : ERRORID
VAR_INPUT
	nParam1 : DINT; //Drops
	nParam2 : DINT; //nicht benutzt
END_VAR

VAR_OUTPUT
	bIsContinous : BOOL;
END_VAR

VAR
	stActionData : ST_ActionData;
END_VAR
IF nParam1 = 0 THEN //DauerDispensen
	bIsContinous := TRUE;
	stActionData.aParams[1] := 0; //Continous
ELSE
	stActionData.aParams[1] := nParam1; //Drops
END_IF

stActionData.eAction := E_Action.ACTION_DispenseDrops;
stActionData.aParams[2] := 1; //On
M_StartUniDispense := M_ExeAction(stActionData);
END_METHOD

METHOD M_StopUniDispense : ERRORID
VAR_INPUT
END_VAR
M_CancelAction(E_Action.ACTION_DispenseDrops);
END_METHOD

PROPERTY P_bSensorMounted : BOOL
GET
IF pParentMzTool^.P_eObjectType = E_ObjectType.OBJECTTYPE_SinglePiezoHolder THEN
	P_bSensorMounted := pZAxisRef^.stInput.nToolState.1;	
END_IF
END_GET
END_PROPERTY

PROPERTY P_nDrypadArea : USINT
GET
P_nDrypadArea := nDrypadArea;
END_GET
END_PROPERTY

PROPERTY P_nObjIdDiluter : UINT
GET
IF pDiluter > 0 THEN
	P_nObjIdDiluter := pDiluter^.P_nObjectID;
END_IF
END_GET
END_PROPERTY

PROPERTY P_nTestResult : UDINT
GET
P_nTestResult := nTestResult;
END_GET
SET
nTestResult := P_nTestResult;
END_SET
END_PROPERTY

PROPERTY P_pDiluter : POINTER TO FB_Diluter
GET
P_pDiluter := pDiluter;
END_GET
END_PROPERTY

PROPERTY P_pPiezoRef : POINTER TO FB_PiezoRef
GET
P_pPiezoRef := pFbPiezoRef;
END_GET
END_PROPERTY

PROPERTY P_rToolRadius : REAL
GET
VAR
	stDim : ST_3DDimension;
END_VAR
P_rToolRadius := 1500.0;
END_GET
END_PROPERTY

PROPERTY P_stCurrentXYArea : FB_RectAngle
GET
VAR
	stPoint : ST_3DPoint;
END_VAR
stPoint := P_stCurrentPosPhys;
P_stCurrentXYArea.X1 := stPoint.X - 1500.0;
P_stCurrentXYArea.X2 := stPoint.X + 1500.0;
P_stCurrentXYArea.Y1 := stPoint.Y - 1500.0;
P_stCurrentXYArea.Y2 := stPoint.Y + 1500.0;
END_GET
END_PROPERTY

PROPERTY P_tDryTime : TIME
GET
P_tDryTime := tDryTime;
END_GET
END_PROPERTY

END_FUNCTION_BLOCK

// ---- Objects/Tools/FB_TitrationTool.TcPOU
FUNCTION_BLOCK FB_TitrationTool EXTENDS FB_MzTool
VAR
	
	stCenterPos: ST_3DPoint;
	stCenterOffset: ST_3DPoint;
	///****************************************Aktionvariablen****************************************************
	///Action: "InitTool"
	bInitTool: BOOL;
	bInitSpecFlag: BOOL := TRUE;
	nStateA_InitTool: USINT;
	timeout: TON;
END_VAR
VAR CONSTANT
	cNumberOfSlots: UINT := 2;
END_VAR

SUPER^();	//FB_MzTool aufrufen

//Prozessdaten aktualisieren
aObjProcData[nNotifyId] := stProcessData;

ACTION A_Reset:
nStateA_ResetSpec := 80;
SUPER^.A_Reset();
END_ACTION

ACTION A_Stop:
IF nStateA_Stop = 0 THEN
	IF bInitTool AND nStateA_InitTool < 70 THEN
		nStateA_InitTool := 70;
	END_IF
	
	nStateA_Stop := 1;
END_IF

SUPER^.A_Stop();
END_ACTION

METHOD FB_init : BOOL
VAR_INPUT
	bInitRetains : BOOL; // if TRUE, the retain variables are initialized (warm start / cold start)
	bInCopyCode : BOOL;  // if TRUE, the instance afterwards gets moved into the copy code (online change)
END_VAR
eObjectType := E_ObjectType.OBJECTTYPE_TitrationTool;
eObjectGroup := E_ObjectGroup.OBJECTGROUP_MzTool OR E_ObjectGroup.OBJECTGROUP_Device;
END_METHOD

METHOD M_AddChild : ERRORID
VAR_INPUT
	pObject : POINTER TO FB_Object;
	nSlotNr	: UINT;
	nIndex 	: INT;
END_VAR
//Kann folgende Objekt-Typen aufnehmen
//pH-Elektrode, PassivPip
IF pObject > 0 THEN
	IF pObject^.P_eObjectType = E_ObjectType.OBJECTTYPE_pHElectrode OR
		pObject^.P_eObjectType = E_ObjectType.OBJECTTYPE_DummyTool OR
		pObject^.P_eObjectType = E_ObjectType.OBJECTTYPE_PassivPip THEN
		M_AddChild := SUPER^.M_AddChild(pObject,nSlotNr,nIndex);
	ELSE
		M_AddChild := E_ErrorIdObjMgmt.ERRORID_InvalidParentObject;
	END_IF
ELSE
	M_AddChild := E_ErrorIdObjMgmt.ERRORID_InvalidParentObject;
END_IF
END_METHOD

METHOD M_CancelAction
VAR_INPUT
	eAction : E_Action;
END_VAR
CASE eAction OF
	(*E_Action.ACTION_Aspirate:
		IF bAspirate AND nStateA_Aspirate < 70 THEN
			nStateA_Aspirate := 70;
		END_IF
	E_Action.ACTION_Dispense:
		IF bDispense AND nStateA_Dispense < 70 THEN
			nStateA_Dispense := 70;
		END_IF
	E_Action.ACTION_DispenseDrops:
		IF bDispensePiezo AND nStateA_DispensePiezo < 70 THEN
			nStateA_DispensePiezo := 70;
		END_IF*)
ELSE
	SUPER^.M_CancelAction(eAction);
END_CASE
END_METHOD

METHOD M_CheckAction : ERRORID
VAR_INPUT
	refActionData	: REFERENCE TO ST_ActionData;
	pCorrelObject	: POINTER TO FB_Object;
END_VAR
VAR
	pTarget : POINTER TO FB_TargetBase;
	pRack	: POINTER TO FB_Rack;
	pSlot	: POINTER TO FB_PieceSlot;	
END_VAR
CASE refActionData.eAction OF
	E_Action.ACTION_InsertTool:
		//TitrationTool darf nur in offene Vials eintauchen
		//-> Target muss also ein VialRack sein
		pTarget := pCorrelObject;
		IF pTarget > 0 THEN
			IF (pTarget^.P_eObjectGroup AND E_ObjectGroup.OBJECTGROUP_Rack) = E_ObjectGroup.OBJECTGROUP_Rack THEN
				pRack := pTarget;
				pSlot := pRack^.M_GetSlot(DINT_TO_UINT(refActionData.aParams[2]));
				IF pSlot > 0 THEN
					IF pSlot^.P_pPiece = 0 THEN
						M_CheckAction := E_ErrorIdCmd.ERRORID_NoPieceInSlot;
						RETURN;
					ELSIF NOT (pSlot^.P_pPiece^.P_eObjectType = E_ObjectType.OBJECTTYPE_Vial OR pSlot^.P_pPiece^.P_eObjectType = E_ObjectType.OBJECTTYPE_FlipTube) THEN
						M_CheckAction := E_ErrorIdCmd.ERRORID_InvalidPieceType;
					END_IF
				ELSE
					M_CheckAction := E_ErrorIdCmd.ERRORID_InvalidTargetSlot;
					RETURN;
				END_IF	
			ELSE
				M_CheckAction := E_ErrorIdCmd.ERRORID_UnsuitableTarget;	
			END_IF
		ELSE
			M_CheckAction := E_ErrorIdCmd.ERRORID_UnsuitableTarget;	
		END_IF	
	E_Action.ACTION_WashTool:
		RETURN;
	E_Action.ACTION_MeasureTool:
		IF fbObjectDirectory.M_GetObjType(refActionData.nTarget) <> E_ObjectType.OBJECTTYPE_TipCalibrator THEN
			M_CheckAction := E_ErrorIdCmd.ERRORID_UnsuitableTarget;
			RETURN;
		END_IF
ELSE
	M_CheckAction := SUPER^.M_CheckAction(refActionData, pCorrelObject);
END_CASE
END_METHOD

METHOD M_GetAllProps : ERRORID
VAR_INPUT
	refCmdData : REFERENCE TO  ST_CmdData;
END_VAR

VAR
	i : UINT;
	pToolSlot	: POINTER TO FB_Slot;
END_VAR
//BaseProperties lesen
SUPER^.M_GetAllProps(refCmdData);
//BaseProperties lesen
nCurrentPropIndex := nCurrentPropIndex + 1;
refCmdData.n32Data[nCurrentPropIndex] := REAL_TO_DINT(stCenterPos.X);
nCurrentPropIndex := nCurrentPropIndex + 1;
refCmdData.n32Data[nCurrentPropIndex] := REAL_TO_DINT(stCenterPos.Y);
nCurrentPropIndex := nCurrentPropIndex + 1;
refCmdData.n32Data[nCurrentPropIndex] := REAL_TO_DINT(stCenterPos.Z);
nCurrentPropIndex := nCurrentPropIndex + 1;
refCmdData.n32Data[nCurrentPropIndex] := REAL_TO_DINT(stCenterOffset.X);
nCurrentPropIndex := nCurrentPropIndex + 1;
refCmdData.n32Data[nCurrentPropIndex] := REAL_TO_DINT(stCenterOffset.Y);
nCurrentPropIndex := nCurrentPropIndex + 1;
refCmdData.n32Data[nCurrentPropIndex] := REAL_TO_DINT(stCenterOffset.Z);
END_METHOD

METHOD M_SetAllProps : ERRORID
VAR_INPUT
	refCmdData : REFERENCE TO  ST_CmdData;
END_VAR

VAR
	nParentMzToolObjId	: UINT;
	pParentTool 		: POINTER TO FB_MzTool;
	pParentHead 		: POINTER TO FB_MzHead;
END_VAR
M_SetAllProps := SUPER^.M_SetAllProps(refCmdData);

IF M_SetAllProps > 0 THEN
	RETURN;
END_IF

//Spezi-Paramter schreiben
nCurrentPropIndex := nCurrentPropIndex + 1;
nSpecPropIndex := nCurrentPropIndex;
stCenterPos.X := DINT_TO_REAL(refCmdData.n32Data[nCurrentPropIndex]);
nCurrentPropIndex := nCurrentPropIndex + 1;
stCenterPos.Y := DINT_TO_REAL(refCmdData.n32Data[nCurrentPropIndex]);
nCurrentPropIndex := nCurrentPropIndex + 1;
stCenterPos.Z := DINT_TO_REAL(refCmdData.n32Data[nCurrentPropIndex]);
nCurrentPropIndex := nCurrentPropIndex + 1;
stCenterOffset.X := DINT_TO_REAL(refCmdData.n32Data[nCurrentPropIndex]);
nCurrentPropIndex := nCurrentPropIndex + 1;
stCenterOffset.Y := DINT_TO_REAL(refCmdData.n32Data[nCurrentPropIndex]);
nCurrentPropIndex := nCurrentPropIndex + 1;
stCenterOffset.Z := DINT_TO_REAL(refCmdData.n32Data[nCurrentPropIndex]);

nNoOfProps := nCurrentPropIndex + 1;
END_METHOD

METHOD M_SetSingleProp : ERRORID
VAR_INPUT
	refCmdData: REFERENCE TO ST_CmdData;
END_VAR
IF nSpecPropIndex = refCmdData.aHeader[1] THEN
	stCenterPos.X := DINT_TO_REAL(refCmdData.n32Data[0]);
ELSIF (nSpecPropIndex + 1) = refCmdData.aHeader[1] THEN
	stCenterPos.Y := DINT_TO_REAL(refCmdData.n32Data[0]);
ELSIF (nSpecPropIndex + 2) = refCmdData.aHeader[1] THEN
	stCenterPos.Z := DINT_TO_REAL(refCmdData.n32Data[0]);
ELSIF (nSpecPropIndex + 3) = refCmdData.aHeader[1] THEN
	stCenterOffset.X := DINT_TO_REAL(refCmdData.n32Data[0]);
ELSIF (nSpecPropIndex + 4) = refCmdData.aHeader[1] THEN
	stCenterOffset.Y := DINT_TO_REAL(refCmdData.n32Data[0]);
ELSIF (nSpecPropIndex + 5) = refCmdData.aHeader[1] THEN
	stCenterOffset.Z := DINT_TO_REAL(refCmdData.n32Data[0]);
ELSE
	M_SetSingleProp := SUPER^.M_SetSingleProp(refCmdData);	
END_IF
END_METHOD

PROPERTY P_rToolRadius : REAL
GET
VAR
	stDim : ST_3DDimension;
END_VAR
P_rToolRadius := 2500.0;
END_GET
END_PROPERTY

PROPERTY P_stAbsPosPhys : ST_3DPoint
GET
VAR
	stTemp: ST_3DPoint;
	stDim: ST_3DDimension;
END_VAR
//Die absolute Postion eines Tool in "Z" hat nicht den gleichen Bezug wie X und Y
//X und Y beziehen sich auf den Koordinatenursprung, wenn die Achsen theoretisch aus Antrieb (0;0) stehen
//Z bezieht sich auf die Sliderunterkante des Z-Antriebes verechnet mit AbsPos vom Head(Ergebnis ist in den meisten Fällen negativ)

stTemp := F_Add3DPoints(stRelPos,stOffset);
//AbsPos vom ParentSlot holen
IF pParentSlot > 0 THEN
	stTemp := F_Add3DPoints(stTemp,pParentSlot^.P_stAbsPos);
END_IF

stTemp := F_Add3DPoints(stTemp,stCenterPos);
P_stAbsPosPhys := F_Add3DPoints(stTemp,stCenterOffset);
END_GET
END_PROPERTY

END_FUNCTION_BLOCK

// ---- Objects/Tools/FB_VermesDisp.TcPOU
FUNCTION_BLOCK FB_VermesDisp EXTENDS FB_GCodeTool
VAR_INPUT
END_VAR
VAR_OUTPUT
END_VAR
VAR
	//Reference zu TripleTrigger
	pPulseTrainChannel : POINTER TO ST_PulseTrainChannel;
	fbPulseTrainControl : FB_PulseTrainControl;

	//Specproperties
	nTriggerChannel		: USINT;
	pPneuChannelPress	: POINTER TO FB_PneuChannelRef;
	nDOutChanValvePress	: USINT;	//Digitaler Ausgangskanal MzHead Druckventil
	nValveNrCool		: USINT;
	
	
	//****************************************Aktionvariablen****************************************************
	
	stActionDataSpec	: ST_ActionData;
	
	//Action: "SetPressure"
	bSetPress			: BOOL;
	fbSetPress			: FB_SetPressure;

	//Action: "Dispense"
	bDispense				: BOOL;
	nStateA_Dispense		: USINT;
	nDrops					: UINT;
	bDispenseStart			: BOOL;
	
END_VAR

IF eCurrentState = E_MachineState.MACHINESTATE_Active THEN

	IF bSetPress THEN
		fbSetPress(pPneuChannelRef:= pPneuChannelPress);
		IF NOT fbSetPress.bBusy THEN
			IF fbSetPress.bError THEN
				bError := TRUE;
				stError.ErrorId := fbSetPress.nErrorId;
				stError.POU := E_POU.POU_FB_VermesDisp;
				fbErrorList.M_Add(stError);
			END_IF
			bSetPress := FALSE;
			fbSetPress(pPneuChannelRef:= pPneuChannelPress, bExecute:= FALSE);
			M_RemoveListEntry(nSearchValue:= E_Action.ACTION_SetPressure);
		END_IF
	END_IF

	IF bDispense THEN
		A_Dispense();
		IF nStateA_Dispense >= 80 THEN
			IF nStateA_Dispense >= 99 THEN
				bError := TRUE;	
			END_IF
			bDispense := FALSE;
			nStateA_Dispense := 0;
			M_RemoveListEntry(nSearchValue:= E_Action.ACTION_DispenseDrops);
		END_IF
	END_IF
END_IF

SUPER^();	//FB_MzTool aufrufen

//Prozessdaten aktualisieren
IF pPneuChannelPress > 0 THEN
	stProcessData.n32Data[7] := pPneuChannelPress^.P_nCurrentPressure;
END_IF

IF pFbMultiZ > 0 THEN
	IF nDOutChanValvePress > 0 AND nDOutChanValvePress < 8 THEN
		stProcessData.n32Data[8] := BOOL_TO_DINT(pFbMultiZ^.aDigiOut[nDOutChanValvePress]);
	END_IF
END_IF
//DispenserStatus
stProcessData.n32Data[9] := BOOL_TO_DINT(fbPulseTrainControl.P_bBusy);

//ValveStatusCool
IF nValveNrCool > 0 THEN
	stProcessData.n32Data[10] := BOOL_TO_DINT(aValves[nValveNrCool].bDigiOut1);
END_IF

aObjProcData[nNotifyId] := stProcessData;

ACTION A_Dispense:
CASE nStateA_Dispense OF
	0:
		fbPulseTrainControl.M_Start(nDrops);
		nStateA_Dispense := 1;

	1:	//Einen Zyklus warten
		nStateA_Dispense := 2;
		
	2:	//Warten bis Dispensen fertig
		IF NOT fbPulseTrainControl.P_bBusy THEN
			fbPulseTrainControl.M_Stop();
			nStateA_Dispense := 80;
		END_IF
		
	70:	//Abbrechen
		fbPulseTrainControl.M_Stop();
		nStateA_Dispense := 80;
END_CASE
END_ACTION

ACTION A_Reset:
//Ist noch eine Aktion aktiv?
IF nStateA_ResetSpec = 0 THEN
	IF bDispense THEN
		bDispense := FALSE;
		nStateA_Dispense := 0;
	END_IF
	
	IF bSetPress THEN
		bSetPress := FALSE;
		fbSetPress(bExecute:= FALSE, pPneuChannelRef:= pPneuChannelPress);
	END_IF
 
	nStateA_ResetSpec := 80;
END_IF

SUPER^.A_Reset();
END_ACTION

ACTION A_Stop:
IF nStateA_Stop = 0 THEN
	
	IF bSetPress THEN
		fbSetPress(bExecute:= FALSE, pPneuChannelRef:= pPneuChannelPress);
	END_IF

	IF bDispense AND nStateA_Dispense < 70 THEN
		nStateA_Dispense := 70;
	END_IF
	
	nStateA_Stop := 1;	
END_IF

SUPER^.A_Stop();
END_ACTION

METHOD FB_init : BOOL
VAR_INPUT
	bInitRetains : BOOL; // if TRUE, the retain variables are initialized (warm start / cold start)
	bInCopyCode : BOOL;  // if TRUE, the instance afterwards gets moved into the copy code (online change)
END_VAR
eObjectType := E_ObjectType.OBJECTTYPE_VermesDisp;
eObjectGroup := E_ObjectGroup.OBJECTGROUP_MzTool OR E_ObjectGroup.OBJECTGROUP_Device;
END_METHOD

METHOD M_AddChild : ERRORID
VAR_INPUT
	pObject : POINTER TO FB_Object;
	nSlotNr	: UINT;
	nIndex 	: INT;
END_VAR
//Kann keine Objekte aufnehmen
M_AddChild := E_ErrorIdObjMgmt.ERRORID_ObjectCanNotTakeChilds;
END_METHOD

METHOD M_CancelAction
VAR_INPUT
	eAction : E_Action;
END_VAR
CASE eAction OF
	E_Action.ACTION_SetPressure:
		IF bSetPress THEN
			fbSetPress(bExecute:= FALSE, pPneuChannelRef:= pPneuChannelPress);
		END_IF
		
	E_Action.ACTION_DispenseDrops:
		IF bDispense AND nStateA_Dispense < 70 THEN
			nStateA_Dispense := 70;
		END_IF
ELSE
	SUPER^.M_CancelAction(eAction);
END_CASE
END_METHOD

METHOD M_CheckAction : ERRORID
VAR_INPUT
	refActionData 	: REFERENCE TO ST_ActionData;
	pCorrelObject	: POINTER TO FB_Object;
END_VAR

VAR
END_VAR
CASE refActionData.eAction OF
	E_Action.ACTION_DispenseDrops, //BasicAction für ActionOnArray
	E_Action.ACTION_TeachTarget:
		RETURN;
ELSE
	M_CheckAction := SUPER^.M_CheckAction(refActionData, pCorrelObject);
END_CASE
END_METHOD

METHOD M_CheckProcDataType : BOOL
VAR_INPUT
	eProcDataType : E_ProcDataType;
END_VAR
IF eProcDataType = E_ProcDataType.PROCDATATYPE_Temp1 THEN
	M_CheckProcDataType := TRUE;
END_IF
END_METHOD

METHOD M_ClearAllProps
VAR_INPUT
	bIgnoreParent : BOOL; //Es wird das gesamte OD gelöscht. -> Zeiger auf Parent nicht mehr gültig!
END_VAR
pPneuChannelPress := 0;
SUPER^.M_ClearAllProps(bIgnoreParent);
END_METHOD

METHOD M_ExeAction : ERRORID
VAR_INPUT
	refActionData : REFERENCE TO ST_ActionData;	
END_VAR
IF NOT (eCurrentState = E_MachineState.MACHINESTATE_Idle OR
	eCurrentState = E_MachineState.MACHINESTATE_Active OR
	eCurrentState = E_MachineState.MACHINESTATE_Ready) THEN
	M_ExeAction := E_ErrorIdCmd.ERRORID_InvalidState;
	RETURN;
END_IF

CASE refActionData.eAction OF
		
	E_Action.ACTION_SetPressure:
		fbSetPress(bExecute:= FALSE, pPneuChannelRef:= pPneuChannelPress); //eventueller Fehler wird auch zurückgesetzt
		fbSetPress.bAwait := DINT_TO_BOOL(refActionData.aParams[1]);
		fbSetPress.nValue := DINT_TO_INT(refActionData.aParams[2]);
		fbSetPress.nTolerancePlus := DINT_TO_INT(refActionData.aParams[3]);
		fbSetPress.nToleranceMinus := DINT_TO_INT(refActionData.aParams[4]);
		fbSetPress.tTimeout := DINT_TO_TIME(refActionData.aParams[5]);
		
		fbSetPress(bExecute:= TRUE,	pPneuChannelRef:= pPneuChannelPress,nErrorId=> M_ExeAction);
		IF fbSetPress.bError THEN
			RETURN;
		END_IF
		
		IF NOT bSetPress AND fbSetPress.bBusy THEN
			bSetPress := TRUE;
			fbList.A_AddHeadValue(hList := hList, putValue := E_Action.ACTION_SetPressure);
		ELSE
			RETURN;	
		END_IF

	E_Action.ACTION_SwitchPressure:
		IF nDOutChanValvePress > 0 AND nDOutChanValvePress < 8 THEN
			IF refActionData.aParams[1] = 1 THEN
				pFbMultiZ^.aDigiOut[nDOutChanValvePress] := TRUE;
			ELSE
				pFbMultiZ^.aDigiOut[nDOutChanValvePress] := FALSE;
			END_IF
		END_IF
		
	E_Action.ACTION_DispenseDrops:
		bDispenseStart := DINT_TO_BOOL(refActionData.aParams[2]);
		IF NOT bDispense AND bDispenseStart THEN
			nDrops := DINT_TO_UINT(refActionData.aParams[1]);
			fbList.A_AddHeadValue( hList := hList, putValue := E_Action.ACTION_DispenseDrops);
			bDispense := TRUE;
		ELSE
			fbPulseTrainControl.M_Stop();
		END_IF
		
	E_Action.ACTION_Cooling:
		IF nValveNrCool > 0 THEN
			IF refActionData.aParams[2] = 1 THEN
				aValves[nValveNrCool].M_On(1);
			ELSE
				aValves[nValveNrCool].M_Off();
			END_IF
		END_IF
	ELSE
		M_ExeAction := SUPER^.M_ExeAction(refActionData);
		RETURN;
END_CASE
bBusy := TRUE;
eCurrentState := E_MachineState.MACHINESTATE_Active;
END_METHOD

METHOD M_GetAllProps : ERRORID
VAR_INPUT
	refCmdData : REFERENCE TO  ST_CmdData;
END_VAR
//BaseProperties lesen
SUPER^.M_GetAllProps(refCmdData);
//BaseProperties lesen
nCurrentPropIndex := nCurrentPropIndex + 1;
refCmdData.n32Data[nCurrentPropIndex] := nTriggerChannel;
nCurrentPropIndex := nCurrentPropIndex + 1;
refCmdData.n32Data[nCurrentPropIndex] := fbPulseTrainControl.M_GetFrequency();
nCurrentPropIndex := nCurrentPropIndex + 1;
refCmdData.n32Data[nCurrentPropIndex] := fbPulseTrainControl.M_GetPulse();

nCurrentPropIndex := nCurrentPropIndex + 1;
IF pPneuChannelPress > 0 THEN
	refCmdData.n32Data[nCurrentPropIndex] := pPneuChannelPress^.nChannel;
ELSE
	refCmdData.n32Data[nCurrentPropIndex] := 0;
END_IF

nCurrentPropIndex := nCurrentPropIndex + 1;
refCmdData.n32Data[nCurrentPropIndex] := nDOutChanValvePress;
nCurrentPropIndex := nCurrentPropIndex + 1;
refCmdData.n32Data[nCurrentPropIndex] := nValveNrCool;
END_METHOD

METHOD M_SetAllProps : ERRORID
VAR_INPUT
	refCmdData : REFERENCE TO  ST_CmdData;
END_VAR

VAR
	nPneuChannel : USINT;
END_VAR
M_SetAllProps := SUPER^.M_SetAllProps(refCmdData);

IF M_SetAllProps > 0 THEN
	RETURN;
END_IF

//TriggerChannel
nCurrentPropIndex := nCurrentPropIndex + 1;
nSpecPropIndex := nCurrentPropIndex;
nTriggerChannel := DINT_TO_USINT(refCmdData.n32Data[nCurrentPropIndex]);
pPulseTrainChannel := aFbIOExpanderRef[1].M_GetPulseTrainChannel(nTriggerChannel);
IF pPulseTrainChannel = 0 THEN
	M_SetAllProps := E_ErrorIdObjMgmt.ERRORID_InvalidTriggerChannel;
	RETURN;	
END_IF

fbPulseTrainControl.M_SetPulseTrainChannel(pPulseTrainChannel);

//Frequenz
nCurrentPropIndex := nCurrentPropIndex + 1;
(*IF NOT (refCmdData.n32Data[nCurrentPropIndex] >= 16 AND refCmdData.n32Data[nCurrentPropIndex] <= 1000000) THEN	
	M_SetAllProps := E_ErrorIdObjMgmt.ERRORID_InvalidFrequency;
	RETURN;
END_IF
pTripleTrigRef^.M_SetFrequency(nTriggerChannel,refCmdData.n32Data[nCurrentPropIndex]);*)
M_SetAllProps := fbPulseTrainControl.M_SetFrequency(DINT_TO_UINT(refCmdData.n32Data[nCurrentPropIndex]));
IF M_SetAllProps > 0 THEN
	RETURN;
END_IF

//Plusbreite
nCurrentPropIndex := nCurrentPropIndex + 1;
(*IF NOT (refCmdData.n32Data[nCurrentPropIndex] >= 0 AND refCmdData.n32Data[nCurrentPropIndex] <= 65535) THEN
	M_SetAllProps := E_ErrorIdObjMgmt.ERRORID_InvalidPulseWidth;  //Error
	RETURN;
END_IF
pTripleTrigRef^.M_SetPulse(nTriggerChannel,DINT_TO_UINT(refCmdData.n32Data[nCurrentPropIndex]));*)
M_SetAllProps := fbPulseTrainControl.M_SetPulse(DINT_TO_UINT(refCmdData.n32Data[nCurrentPropIndex]));
IF M_SetAllProps > 0 THEN
	RETURN;
END_IF

//PneuChannel Druck
nCurrentPropIndex := nCurrentPropIndex + 1;
nPneuChannel := DINT_TO_USINT(refCmdData.n32Data[nCurrentPropIndex]);
IF NOT (nPneuChannel >= 0 AND nPneuChannel <= cNoOfPneuChannels) THEN
	M_SetAllProps := E_ErrorIdObjMgmt.ERRORID_InvalidPneuChannel;
	RETURN;	
END_IF
pPneuChannelPress := ADR(aFbPneuChannel[nPneuChannel]);

//digitaler Ausgang Kopfbasisplatine Druckventil am Kopf
nCurrentPropIndex := nCurrentPropIndex + 1;
nDOutChanValvePress := DINT_TO_USINT(refCmdData.n32Data[nCurrentPropIndex]);	//Digitaler Ausgangskanal MzHead Druckventil
IF NOT (nDOutChanValvePress >= 0 AND nDOutChanValvePress <= 7) THEN
	M_SetAllProps := E_ErrorIdObjMgmt.ERRORID_InvalidMzDOutChannel;
	RETURN;	
END_IF

//Ventilnummer in FBox für Druckluftkühlung
nCurrentPropIndex := nCurrentPropIndex + 1;
nValveNrCool := DINT_TO_USINT(refCmdData.n32Data[nCurrentPropIndex]);
IF NOT (nValveNrCool >= 0 AND nValveNrCool <= cNoOfValves) THEN
	M_SetAllProps := E_ErrorIdObjMgmt.ERRORID_InvalidValveNumber;
	RETURN;	
END_IF

nNoOfProps := nCurrentPropIndex + 1;
END_METHOD

METHOD M_SetSingleProp : ERRORID
VAR_INPUT
	refCmdData : REFERENCE TO  ST_CmdData;
END_VAR
IF nSpecPropIndex = refCmdData.aHeader[1] THEN
	IF refCmdData.n32Data[0] >= 1 AND refCmdData.n32Data[0] <= 3 THEN
		nTriggerChannel := DINT_TO_USINT(refCmdData.n32Data[0]);
		pPulseTrainChannel := aFbIOExpanderRef[1].M_GetPulseTrainChannel(nTriggerChannel);
		IF pPulseTrainChannel > 0 THEN
			fbPulseTrainControl.M_Stop();
			fbPulseTrainControl.M_SetPulseTrainChannel(pPulseTrainChannel);		
		END_IF
	ELSE
		M_SetSingleProp := E_ErrorIdObjMgmt.ERRORID_InvalidTriggerChannel;
		RETURN;
	END_IF
ELSIF (nSpecPropIndex + 1) = refCmdData.aHeader[1] THEN	//Frequenz
	M_SetSingleProp := fbPulseTrainControl.M_SetFrequency(DINT_TO_UINT(refCmdData.n32Data[0]));
ELSIF (nSpecPropIndex + 2) = refCmdData.aHeader[1] THEN //Pulsbreite
	IF NOT (refCmdData.n32Data[0] >= 0 AND refCmdData.n32Data[0] < 65535) THEN
		M_SetSingleProp := E_ErrorIdObjMgmt.ERRORID_InvalidPulseWidth;
		RETURN;
	END_IF
	M_SetSingleProp := fbPulseTrainControl.M_SetPulse(DINT_TO_UINT(refCmdData.n32Data[0]));
ELSE
	M_SetSingleProp := SUPER^.M_SetSingleProp(refCmdData);
END_IF
END_METHOD

METHOD M_StartUniDispense : ERRORID
VAR_INPUT
	nParam1 : DINT; //Drops
	nParam2 : DINT; //nicht benutzt
END_VAR

VAR_OUTPUT
	bIsContinous : BOOL;
END_VAR

VAR
	stActionData : ST_ActionData;
END_VAR
IF nParam1 = 0 THEN //DauerDispensen
	bIsContinous := TRUE;
	stActionData.aParams[1] := 0; //Continous
ELSE
	stActionData.aParams[1] := nParam1; //Drops
END_IF

stActionData.eAction := E_Action.ACTION_DispenseDrops;
stActionData.aParams[2] := 1; //On
M_StartUniDispense := M_ExeAction(stActionData);
END_METHOD

METHOD M_StopUniDispense : ERRORID
VAR_INPUT
END_VAR
M_CancelAction(E_Action.ACTION_DispenseDrops);
END_METHOD

END_FUNCTION_BLOCK

// ---- Hardware/IOExpander/FB_PulseTrainControl.TcPOU
FUNCTION_BLOCK FB_PulseTrainControl
VAR_INPUT
END_VAR
VAR_OUTPUT
END_VAR
VAR
	pPulseTrainChannel : POINTER TO ST_PulseTrainChannel;
	nFrequency : UINT;
END_VAR

METHOD M_GetFrequency : UINT
VAR_INPUT
END_VAR
M_GetFrequency := nFrequency;
END_METHOD

METHOD M_GetPulse : UINT
VAR_INPUT
END_VAR
IF pPulseTrainChannel > 0 THEN
	M_GetPulse := pPulseTrainChannel^.nPulse;
END_IF
END_METHOD

METHOD M_SetFrequency : ERRORID
VAR_INPUT
	nValue : UINT;
END_VAR
IF pPulseTrainChannel = 0 THEN
	M_SetFrequency := E_ErrorIdObjMgmt.ERRORID_InvalidTriggerChannel;
	RETURN;
END_IF
IF nValue >= 16 AND nValue <= 10000 THEN
	nFrequency := nValue;
	pPulseTrainChannel^.nPeriod := UDINT_TO_UINT(1000000 / nFrequency);
ELSE
	M_SetFrequency := E_ErrorIdObjMgmt.ERRORID_InvalidFrequency;
END_IF
END_METHOD

METHOD M_SetPulse : ERRORID
VAR_INPUT
	nValue : UINT;
END_VAR
IF pPulseTrainChannel = 0 THEN
	M_SetPulse := E_ErrorIdObjMgmt.ERRORID_InvalidTriggerChannel;
	RETURN;
END_IF
IF nValue > 0 AND nValue <= 65635 THEN
	pPulseTrainChannel^.nPulse := nValue;
ELSE
	M_SetPulse := E_ErrorIdObjMgmt.ERRORID_InvalidPulseWidth;
END_IF
END_METHOD

METHOD M_SetPulseTrainChannel
VAR_INPUT
	pPulseTrainChannel : POINTER TO ST_PulseTrainChannel;
END_VAR
THIS^.pPulseTrainChannel := pPulseTrainChannel;
END_METHOD

METHOD M_Start
VAR_INPUT
	nNrOfPulses : UINT;
END_VAR
IF pPulseTrainChannel > 0 THEN
	pPulseTrainChannel^.nNoOfPulses := nNrOfPulses;
	pPulseTrainChannel^.nCtrl := 1;
END_IF
END_METHOD

METHOD M_Stop
VAR_INPUT
END_VAR
IF pPulseTrainChannel > 0 THEN
	pPulseTrainChannel^.nCtrl := 0;
END_IF
END_METHOD

PROPERTY P_bBusy : BOOL
GET
IF pPulseTrainChannel > 0 THEN
	P_bBusy := pPulseTrainChannel^.nState.0;
END_IF
END_GET
END_PROPERTY

END_FUNCTION_BLOCK

// ---- Objects/Tools/FB_DummyTool.TcPOU
FUNCTION_BLOCK FB_DummyTool EXTENDS FB_MzTool
VAR_INPUT
END_VAR
VAR_OUTPUT
END_VAR

SUPER^();	//FB_MzTool aufrufen
aObjProcData[nNotifyId] := stProcessData;

ACTION A_Reset:
//Ist noch eine Aktion aktiv?
IF nStateA_ResetSpec = 0 THEN 
	nStateA_ResetSpec := 80;
END_IF

SUPER^.A_Reset();
END_ACTION

METHOD FB_init : BOOL
VAR_INPUT
	bInitRetains : BOOL; // if TRUE, the retain variables are initialized (warm start / cold start)
	bInCopyCode : BOOL;  // if TRUE, the instance afterwards gets moved into the copy code (online change)
END_VAR
eObjectType := E_ObjectType.OBJECTTYPE_DummyTool;
eObjectGroup := E_ObjectGroup.OBJECTGROUP_MzTool OR E_ObjectGroup.OBJECTGROUP_Device;
END_METHOD

END_FUNCTION_BLOCK

// ---- Objects/Tools/FB_Gripper.TcPOU
FUNCTION_BLOCK FB_Gripper EXTENDS FB_MzTool
VAR_INPUT
END_VAR
VAR_OUTPUT
END_VAR
VAR
	//SpecProperties
	pGripperRef	: POINTER TO FB_GripperRef;

	//****************************************Aktionvariablen****************************************************
	
	//Action: "OpenClose"
	bOpenClose			: BOOL;
	nStateA_OpenClose	: USINT;	//Statemachine von A_OpenClose();
	eOpClCtrl			: E_OpClCtrl;
	timerOpenClose 		: TON;
	bCloseWithPiece		: BOOL;		//Dient zur Überwachung, ob bei Schließen wirklich ein Piece geklemmt wird (Position zwischen beiden Endlagen)
END_VAR

IF eCurrentState = E_MachineState.MACHINESTATE_Active THEN
	IF bOpenClose THEN
		A_OpenClose();
		IF nStateA_OpenClose >= 80 THEN
			IF nStateA_OpenClose >= 99 THEN
				bError := TRUE;	
			END_IF
			bOpenClose := FALSE;
			nStateA_OpenClose := 0;
			M_RemoveListEntry(nSearchValue:= E_Action.ACTION_OpenClose);
		END_IF
	END_IF		
END_IF

SUPER^();	//FB_MzTool aufrufen

//Prozessdaten aktualisieren
stProcessData.n32Data[7] := pGripperRef^.P_eGripperState;
aObjProcData[nNotifyId] := stProcessData;

ACTION A_OpenClose:
IF nStateA_OpenClose = 0 THEN
	pGripperRef^.M_Actuate(eOpClCtrl);
	timerOpenClose(IN:= TRUE, PT:= T#500MS);
	nStateA_OpenClose := 1;
ELSIF nStateA_OpenClose = 1 THEN
	timerOpenClose();
	IF timerOpenClose.Q THEN
		timerOpenClose(IN:= FALSE);
		//Auf State checken
		IF eOpClCtrl = E_OpClCtrl.Open THEN
			IF pGripperRef^.P_eGripperState = E_GripperState.Open THEN
				nStateA_OpenClose := 80;
			ELSE
				//Fehler: nicht vollständig geöffnet
				stError.ErrorId := E_ErrorIdCmd.ERRORID_NotFullyOpened;
				nStateA_OpenClose := 99;
			END_IF
		ELSE //Close , hier wird noch unterschieden, ob Soll-State nur HalfClosed sein soll (wird nur bei ExeActionDirect gesetzt)
			IF bCloseWithPiece THEN
				IF pGripperRef^.P_eGripperState = E_GripperState.HalfClosed THEN
					nStateA_OpenClose := 80;
				ELSE
					//Fehler: kein Vial im Gripper
					stError.ErrorId := E_ErrorIdCmd.ERRORID_NoPieceTaken;
					nStateA_OpenClose := 99;
				END_IF
			ELSE //Hier ist nicht eindeutig angeben, ob mit oder ohne Piece (bei manueller Betätigung)
				//In diesem Fall darf der State HalfClosed  oder auch FullyClosed sein.
				IF pGripperRef^.P_eGripperState = E_GripperState.HalfClosed
						OR pGripperRef^.P_eGripperState = E_GripperState.FullyClosed THEN
					nStateA_OpenClose := 80;
				ELSE
					//Fehler beim Schließen des Grippers
					stError.ErrorId := E_ErrorIdCmd.ERRORID_NotFullyClosed;
					nStateA_OpenClose := 99;
				END_IF
			END_IF
		END_IF
	END_IF
END_IF

IF nStateA_OpenClose = 99 THEN
	stError.Cmd := E_Action.ACTION_OpenClose;
	stError.POU := E_POU.POU_FB_Gripper;
	stError.POUAction := E_POUACT.POUACT_A_OpenClose;
	fbErrorList.M_Add(stError);
END_IF
END_ACTION

ACTION A_Reset:
//Ist noch eine Aktion aktiv?
IF nStateA_ResetSpec = 0 THEN 
	nStateA_ResetSpec := 80;
END_IF

SUPER^.A_Reset();
END_ACTION

ACTION A_Stop:
IF nStateA_Stop = 0 THEN
	nStateA_Stop := 1;
END_IF

SUPER^.A_Stop();
END_ACTION

METHOD FB_init : BOOL
VAR_INPUT
	bInitRetains : BOOL; // if TRUE, the retain variables are initialized (warm start / cold start)
	bInCopyCode : BOOL;  // if TRUE, the instance afterwards gets moved into the copy code (online change)
END_VAR
eObjectType := E_ObjectType.OBJECTTYPE_Gripper;
eObjectGroup := E_ObjectGroup.OBJECTGROUP_MzTool OR E_ObjectGroup.OBJECTGROUP_Device;
END_METHOD

METHOD M_AddChild : ERRORID
VAR_INPUT
	pObject : POINTER TO FB_Object;
	nSlotNr	: UINT;
	nIndex 	: INT;	
END_VAR
//Kann folgende Objekt-Typen aufnehmen
//Vial
IF pObject > 0 THEN
	IF pObject^.P_eObjectType = E_ObjectType.OBJECTTYPE_Vial THEN
		M_AddChild := SUPER^.M_AddChild(pObject,nSlotNr,nIndex);
	ELSE
		M_AddChild := E_ErrorIdObjMgmt.ERRORID_InvalidParentObject;
	END_IF
ELSE
	M_AddChild := E_ErrorIdObjMgmt.ERRORID_InvalidParentObject;
END_IF
END_METHOD

METHOD M_CheckAction : ERRORID
VAR_INPUT
	refActionData 	: REFERENCE TO ST_ActionData;
	pCorrelObject	: POINTER TO FB_Object;
END_VAR

VAR
	pRack 			: POINTER TO FB_Rack;
	pReactor 		: POINTER TO FB_Reactor;
	pPowderStation 	: POINTER TO FB_PowderStation;
	pSlot 			: POINTER TO FB_PieceSlot;
	pTarget 		: POINTER TO FB_TargetBase;
END_VAR
CASE refActionData.eAction OF
	E_Action.ACTION_ExchangePiece:
		pTarget := fbObjectDirectory.M_GetObjPointer(refActionData.nTarget);
		//Welches Piece soll gehandelt werden?
		IF refActionData.aParams[2] = 0 THEN //Drop
			IF pPiece = 0 THEN
				M_CheckAction := E_ErrorIdCmd.ERRORID_NoPieceOnTool;
				RETURN;	
			END_IF
			//Gripper kann folgende Pieces handeln
			//Vial, ???
			IF pPiece^.P_eObjectType = E_ObjectType.OBJECTTYPE_Vial THEN
				//Target muss VialRack oder Reaktor sein
				IF pTarget^.P_eObjectType = E_ObjectType.OBJECTTYPE_VialRack THEN
					pRack := pTarget;
					//Slot muss frei sein
					pSlot := pRack^.M_GetSlot(DINT_TO_UINT(refActionData.aParams[1]));
					IF pSlot = 0 THEN
						M_CheckAction := E_ErrorIdCmd.ERRORID_InvalidTargetSlot;
						RETURN;
					ELSIF pSlot^.P_pPiece > 0 THEN
						M_CheckAction := E_ErrorIdCmd.ERRORID_PieceAlreadyInSlot;
						RETURN;
					END_IF
				ELSIF pTarget^.P_eObjectType = E_ObjectType.OBJECTTYPE_Reactor THEN
					//Slot muss frei sein
					pReactor := pTarget;
					IF pReactor^.P_pVial > 0 THEN
						M_CheckAction := E_ErrorIdCmd.ERRORID_PieceAlreadyInSlot;
						RETURN;
					END_IF
				ELSIF pTarget^.P_eObjectType = E_ObjectType.OBJECTTYPE_PowderStation THEN
					//Slot muss frei sein
					pPowderStation := pTarget;
					IF pPowderStation^.P_pVial > 0 THEN
						M_CheckAction := E_ErrorIdCmd.ERRORID_PieceAlreadyInSlot;
						RETURN;
					END_IF
				ELSE
					M_CheckAction := E_ErrorIdCmd.ERRORID_UnsuitableTarget;
					RETURN;
				END_IF
			ELSE
				M_CheckAction := E_ErrorIdCmd.ERRORID_InvalidPieceType;
				RETURN;
			END_IF
		ELSE  //Take
			//Schon ein Piece am Tool?
			IF THIS^.pPiece > 0 THEN
				M_CheckAction := E_ErrorIdCmd.ERRORID_PieceAlreadyOnTool;
				RETURN;
			END_IF
			
			IF pTarget^.P_eObjectType = E_ObjectType.OBJECTTYPE_Reactor THEN
				//Hier kann ein Vial geholt werden
				pReactor := pTarget;
				IF pReactor^.P_pVial = 0 THEN
					M_CheckAction := E_ErrorIdCmd.ERRORID_NoPieceInSlot;
					RETURN;
				ELSIF pReactor^.P_pVial^.P_pSeptum > 0 THEN
					M_CheckAction := E_ErrorIdCmd.ERRORID_SeptumAlreadyOnVial;
					RETURN;
				END_IF
			ELSIF pTarget^.P_eObjectType = E_ObjectType.OBJECTTYPE_PowderStation THEN
				pPowderStation := pTarget;
				IF pPowderStation^.P_pVial = 0 THEN
					M_CheckAction := E_ErrorIdCmd.ERRORID_NoPieceInSlot;
					RETURN;
				END_IF
			ELSIF pTarget^.P_eObjectType = E_ObjectType.OBJECTTYPE_VialRack THEN
				//Hier kann ein Vial geholt werden
				pRack := pTarget;
				pSlot := pRack^.M_GetSlot(DINT_TO_UINT(refActionData.aParams[1]));
				IF pSlot > 0 THEN
					IF pSlot^.P_pPiece = 0 THEN
						M_CheckAction := E_ErrorIdCmd.ERRORID_NoPieceInSlot;
						RETURN;
					ELSIF pSlot^.P_pPiece^.P_eObjectType <> E_ObjectType.OBJECTTYPE_Vial THEN
						M_CheckAction := E_ErrorIdCmd.ERRORID_InvalidPieceType;
						RETURN;
					END_IF
				ELSE
					M_CheckAction := E_ErrorIdCmd.ERRORID_InvalidTargetSlot;
					RETURN;				
				END_IF
			ELSE
				M_CheckAction := E_ErrorIdCmd.ERRORID_UnsuitableTarget;
				RETURN;
			END_IF
		END_IF	
ELSE
	M_CheckAction := SUPER^.M_CheckAction(refActionData, pCorrelObject);
END_CASE
END_METHOD

METHOD M_ExeAction : ERRORID
VAR_INPUT
	refActionData : REFERENCE TO ST_ActionData;	
END_VAR
IF NOT (eCurrentState = E_MachineState.MACHINESTATE_Idle OR
	eCurrentState = E_MachineState.MACHINESTATE_Active OR
	eCurrentState = E_MachineState.MACHINESTATE_Ready) THEN
	M_ExeAction := E_ErrorIdCmd.ERRORID_InvalidState;
	RETURN;
END_IF

IF refActionData.eAction = E_Action.ACTION_OpenClose THEN
	IF NOT bOpenClose THEN
		eOpClCtrl := DINT_TO_USINT(refActionData.aParams[1]);
		fbList.A_AddHeadValue(hList := hList, putValue:= E_Action.ACTION_OpenClose);
		bOpenClose := TRUE;
	ELSE
		RETURN;
	END_IF
 
ELSE
	M_ExeAction := SUPER^.M_ExeAction(refActionData);
	RETURN;
END_IF

bBusy := TRUE;
eCurrentState := E_MachineState.MACHINESTATE_Active;
END_METHOD

METHOD M_OpenClose : ERRORID
VAR_INPUT
	eCtrl			: E_OpClCtrl;
	bCloseWithPiece : BOOL;
END_VAR
IF NOT (eCurrentState = E_MachineState.MACHINESTATE_Idle OR
	eCurrentState = E_MachineState.MACHINESTATE_Active OR
	eCurrentState = E_MachineState.MACHINESTATE_Ready) THEN
	M_OpenClose := E_ErrorIdCmd.ERRORID_InvalidState;
	RETURN;
END_IF

